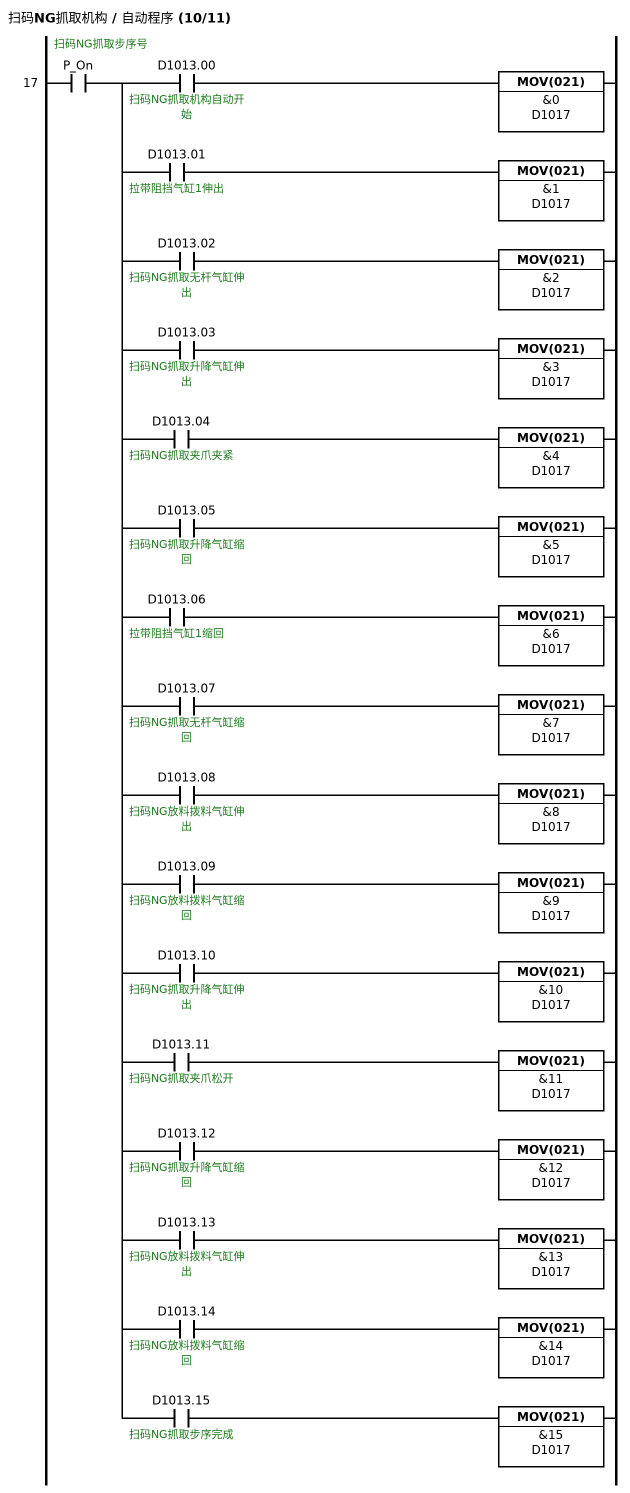
; rung 17: 扫码NG抓取步序号
LD P_On
OUT TR0
AND D1013.00  ; 扫码NG抓取机构自动开始
MOV(021) &0 D1017
LD TR0
AND D1013.01  ; 拉带阻挡气缸1伸出
MOV(021) &1 D1017
LD TR0
AND D1013.02  ; 扫码NG抓取无杆气缸伸出
MOV(021) &2 D1017
LD TR0
AND D1013.03  ; 扫码NG抓取升降气缸伸出
MOV(021) &3 D1017
LD TR0
AND D1013.04  ; 扫码NG抓取夹爪夹紧
MOV(021) &4 D1017
LD TR0
AND D1013.05  ; 扫码NG抓取升降气缸缩回
MOV(021) &5 D1017
LD TR0
AND D1013.06  ; 拉带阻挡气缸1缩回
MOV(021) &6 D1017
LD TR0
AND D1013.07  ; 扫码NG抓取无杆气缸缩回
MOV(021) &7 D1017
LD TR0
AND D1013.08  ; 扫码NG放料拨料气缸伸出
MOV(021) &8 D1017
LD TR0
AND D1013.09  ; 扫码NG放料拨料气缸缩回
MOV(021) &9 D1017
LD TR0
AND D1013.10  ; 扫码NG抓取升降气缸伸出
MOV(021) &10 D1017
LD TR0
AND D1013.11  ; 扫码NG抓取夹爪松开
MOV(021) &11 D1017
LD TR0
AND D1013.12  ; 扫码NG抓取升降气缸缩回
MOV(021) &12 D1017
LD TR0
AND D1013.13  ; 扫码NG放料拨料气缸伸出
MOV(021) &13 D1017
LD TR0
AND D1013.14  ; 扫码NG放料拨料气缸缩回
MOV(021) &14 D1017
LD TR0
AND D1013.15  ; 扫码NG抓取步序完成
MOV(021) &15 D1017

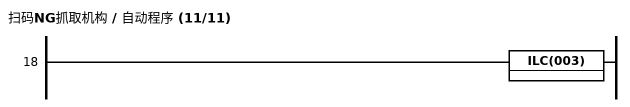
; rung 18
ILC(003)

### Section 状态指示灯

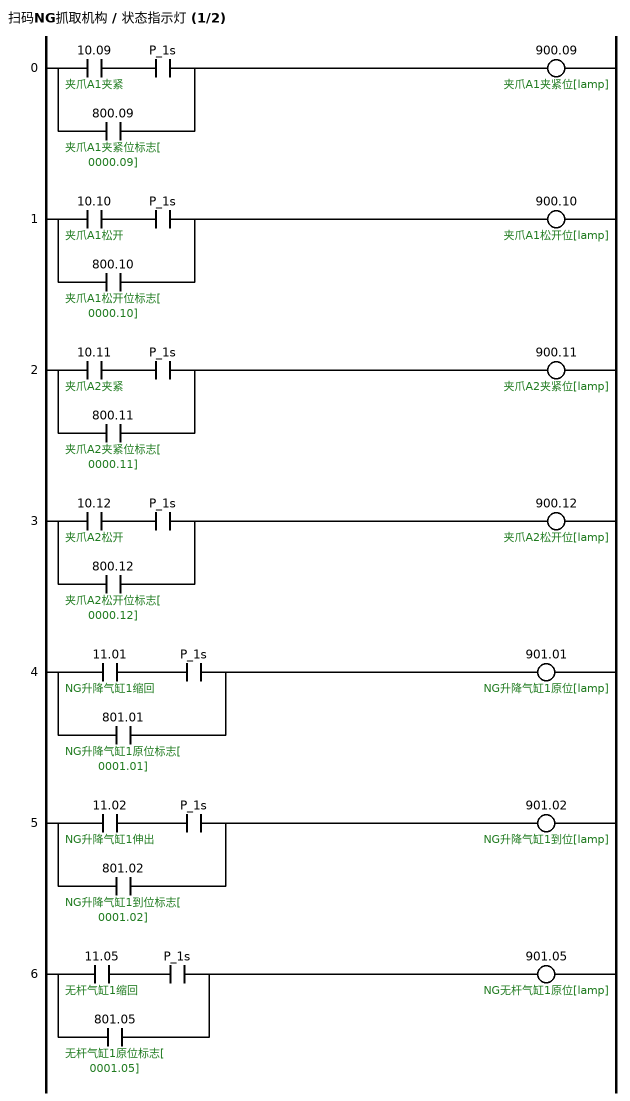
; rung 0
LD 10.09  ; 夹爪A1夹紧
AND P_1s
OR 800.09  ; 夹爪A1夹紧位标志[0000.09]
OUT 900.09  ; 夹爪A1夹紧位[lamp]
; rung 1
LD 10.10  ; 夹爪A1松开
AND P_1s
OR 800.10  ; 夹爪A1松开位标志[0000.10]
OUT 900.10  ; 夹爪A1松开位[lamp]
; rung 2
LD 10.11  ; 夹爪A2夹紧
AND P_1s
OR 800.11  ; 夹爪A2夹紧位标志[0000.11]
OUT 900.11  ; 夹爪A2夹紧位[lamp]
; rung 3
LD 10.12  ; 夹爪A2松开
AND P_1s
OR 800.12  ; 夹爪A2松开位标志[0000.12]
OUT 900.12  ; 夹爪A2松开位[lamp]
; rung 4
LD 11.01  ; NG升降气缸1缩回
AND P_1s
OR 801.01  ; NG升降气缸1原位标志[0001.01]
OUT 901.01  ; NG升降气缸1原位[lamp]
; rung 5
LD 11.02  ; NG升降气缸1伸出
AND P_1s
OR 801.02  ; NG升降气缸1到位标志[0001.02]
OUT 901.02  ; NG升降气缸1到位[lamp]
; rung 6
LD 11.05  ; 无杆气缸1缩回
AND P_1s
OR 801.05  ; 无杆气缸1原位标志[0001.05]
OUT 901.05  ; NG无杆气缸1原位[lamp]

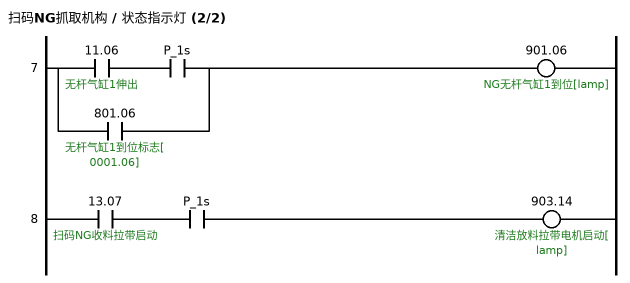
; rung 7
LD 11.06  ; 无杆气缸1伸出
AND P_1s
OR 801.06  ; 无杆气缸1到位标志[0001.06]
OUT 901.06  ; NG无杆气缸1到位[lamp]
; rung 8
LD 13.07  ; 扫码NG收料拉带启动
AND P_1s
OUT 903.14  ; 清洁放料拉带电机启动[lamp]

### Section 输出程序

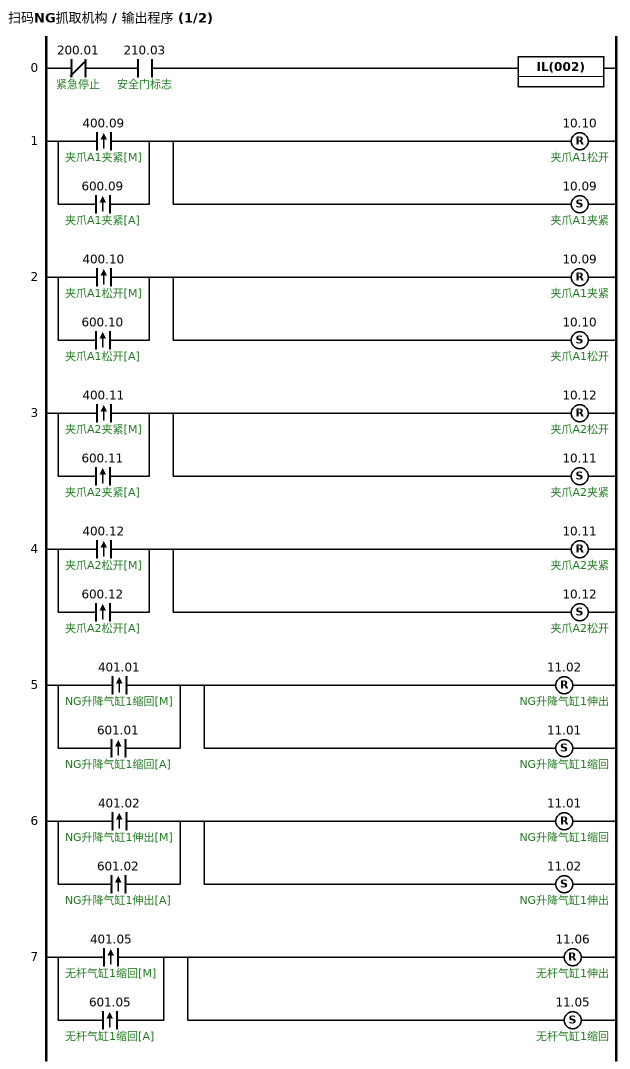
; rung 0
LDNOT 200.01  ; 紧急停止
AND 210.03  ; 安全门标志
IL(002)
; rung 1
@LD 400.09  ; 夹爪A1夹紧[M]
@OR 600.09  ; 夹爪A1夹紧[A]
RSET 10.10  ; 夹爪A1松开
SET 10.09  ; 夹爪A1夹紧
; rung 2
@LD 400.10  ; 夹爪A1松开[M]
@OR 600.10  ; 夹爪A1松开[A]
RSET 10.09  ; 夹爪A1夹紧
SET 10.10  ; 夹爪A1松开
; rung 3
@LD 400.11  ; 夹爪A2夹紧[M]
@OR 600.11  ; 夹爪A2夹紧[A]
RSET 10.12  ; 夹爪A2松开
SET 10.11  ; 夹爪A2夹紧
; rung 4
@LD 400.12  ; 夹爪A2松开[M]
@OR 600.12  ; 夹爪A2松开[A]
RSET 10.11  ; 夹爪A2夹紧
SET 10.12  ; 夹爪A2松开
; rung 5
@LD 401.01  ; NG升降气缸1缩回[M]
@OR 601.01  ; NG升降气缸1缩回[A]
RSET 11.02  ; NG升降气缸1伸出
SET 11.01  ; NG升降气缸1缩回
; rung 6
@LD 401.02  ; NG升降气缸1伸出[M]
@OR 601.02  ; NG升降气缸1伸出[A]
RSET 11.01  ; NG升降气缸1缩回
SET 11.02  ; NG升降气缸1伸出
; rung 7
@LD 401.05  ; 无杆气缸1缩回[M]
@OR 601.05  ; 无杆气缸1缩回[A]
RSET 11.06  ; 无杆气缸1伸出
SET 11.05  ; 无杆气缸1缩回

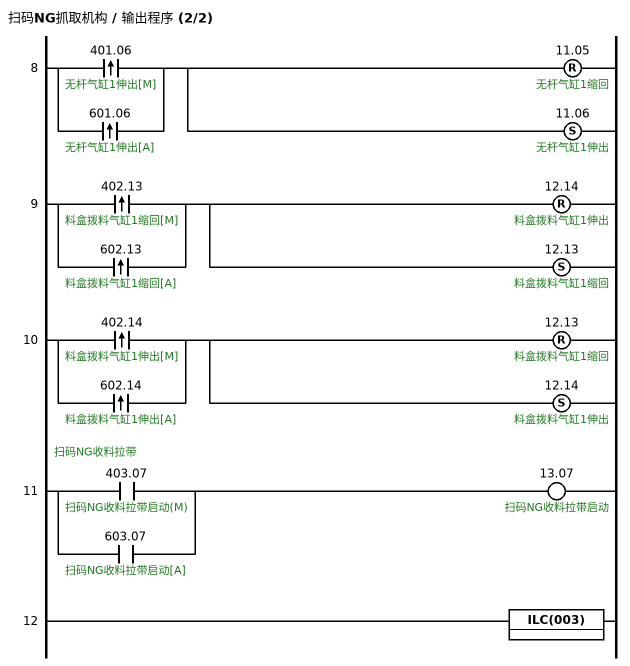
; rung 8
@LD 401.06  ; 无杆气缸1伸出[M]
@OR 601.06  ; 无杆气缸1伸出[A]
RSET 11.05  ; 无杆气缸1缩回
SET 11.06  ; 无杆气缸1伸出
; rung 9
@LD 402.13  ; 料盒拨料气缸1缩回[M]
@OR 602.13  ; 料盒拨料气缸1缩回[A]
RSET 12.14  ; 料盒拨料气缸1伸出
SET 12.13  ; 料盒拨料气缸1缩回
; rung 10
@LD 402.14  ; 料盒拨料气缸1伸出[M]
@OR 602.14  ; 料盒拨料气缸1伸出[A]
RSET 12.13  ; 料盒拨料气缸1缩回
SET 12.14  ; 料盒拨料气缸1伸出
; rung 11: 扫码NG收料拉带
LD 403.07  ; 扫码NG收料拉带启动(M)
OR 603.07  ; 扫码NG收料拉带启动[A]
OUT 13.07  ; 扫码NG收料拉带启动
; rung 12
ILC(003)

### Section END
; rung 0
END(001)

## Program 电池清洁机构 (cyclic task 3)

### Section 主程序

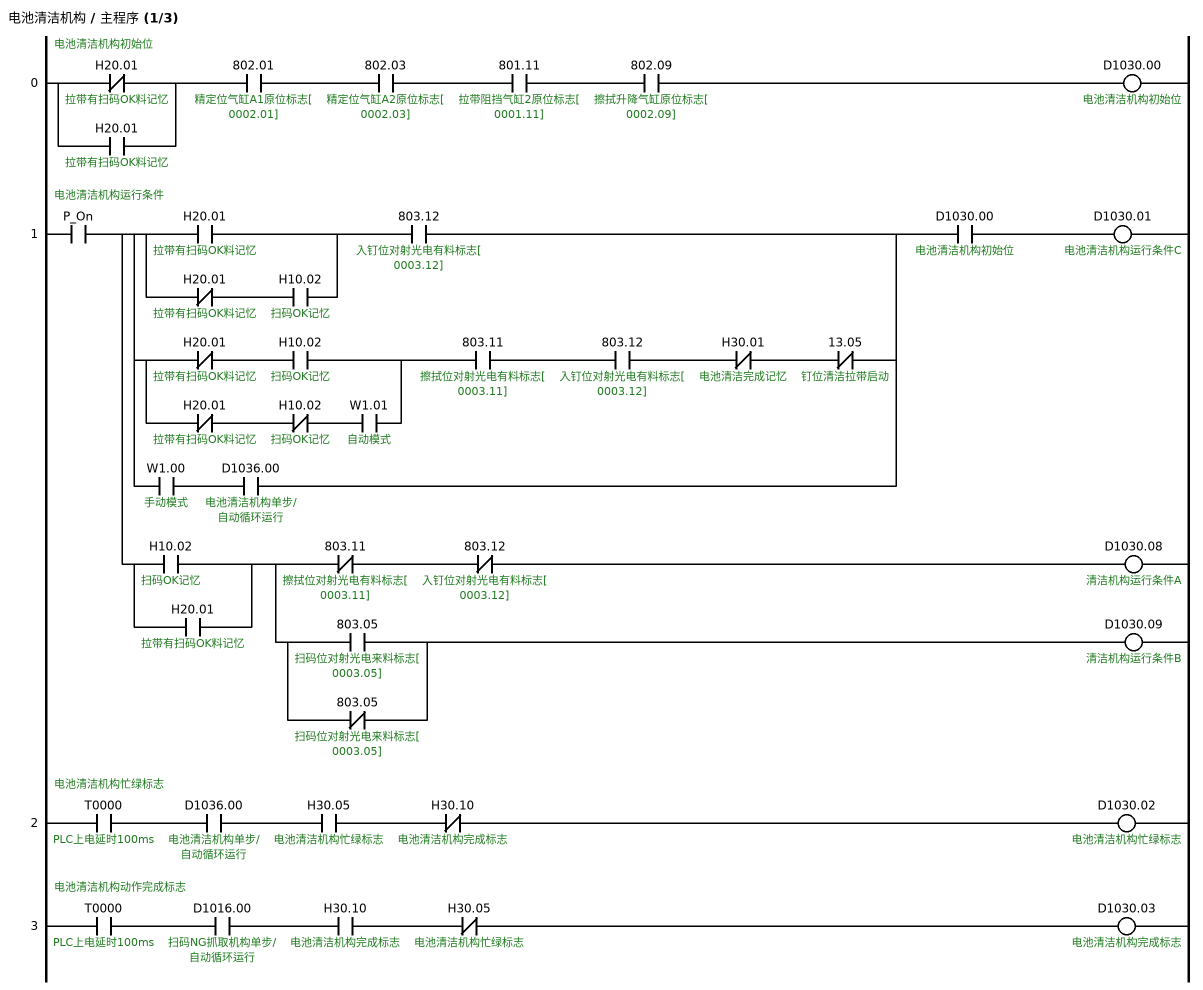
; rung 0: 电池清洁机构初始位
LDNOT H20.01  ; 拉带有扫码OK料记忆
OR H20.01  ; 拉带有扫码OK料记忆
AND 802.01  ; 精定位气缸A1原位标志[0002.01]
AND 802.03  ; 精定位气缸A2原位标志[0002.03]
AND 801.11  ; 拉带阻挡气缸2原位标志[0001.11]
AND 802.09  ; 擦拭升降气缸原位标志[0002.09]
OUT D1030.00  ; 电池清洁机构初始位
; rung 1: 电池清洁机构运行条件
LD P_On
OUT TR0
LD H20.01  ; 拉带有扫码OK料记忆
LDNOT H20.01  ; 拉带有扫码OK料记忆
AND H10.02  ; 扫码OK记忆
ORLD
AND 803.12  ; 入钉位对射光电有料标志[0003.12]
LDNOT H20.01  ; 拉带有扫码OK料记忆
AND H10.02  ; 扫码OK记忆
LDNOT H20.01  ; 拉带有扫码OK料记忆
ANDNOT H10.02  ; 扫码OK记忆
AND W1.01  ; 自动模式
ORLD
AND 803.11  ; 擦拭位对射光电有料标志[0003.11]
AND 803.12  ; 入钉位对射光电有料标志[0003.12]
ANDNOT H30.01  ; 电池清洁完成记忆
ANDNOT 13.05  ; 钉位清洁拉带启动
ORLD
LD W1.00  ; 手动模式
AND D1036.00  ; 电池清洁机构单步/自动循环运行
ORLD
ANDLD
AND D1030.00  ; 电池清洁机构初始位
OUT D1030.01  ; 电池清洁机构运行条件C
LD TR0
LD H10.02  ; 扫码OK记忆
OR H20.01  ; 拉带有扫码OK料记忆
ANDLD
OUT TR0
ANDNOT 803.11  ; 擦拭位对射光电有料标志[0003.11]
ANDNOT 803.12  ; 入钉位对射光电有料标志[0003.12]
OUT D1030.08  ; 清洁机构运行条件A
LD TR0
LD 803.05  ; 扫码位对射光电来料标志[0003.05]
ORNOT 803.05  ; 扫码位对射光电来料标志[0003.05]
ANDLD
OUT D1030.09  ; 清洁机构运行条件B
; rung 2: 电池清洁机构忙绿标志
LD T0000  ; PLC上电延时100ms
AND D1036.00  ; 电池清洁机构单步/自动循环运行
AND H30.05  ; 电池清洁机构忙绿标志
ANDNOT H30.10  ; 电池清洁机构完成标志
OUT D1030.02  ; 电池清洁机构忙绿标志
; rung 3: 电池清洁机构动作完成标志
LD T0000  ; PLC上电延时100ms
AND D1016.00  ; 扫码NG抓取机构单步/自动循环运行
AND H30.10  ; 电池清洁机构完成标志
ANDNOT H30.05  ; 电池清洁机构忙绿标志
OUT D1030.03  ; 电池清洁机构完成标志

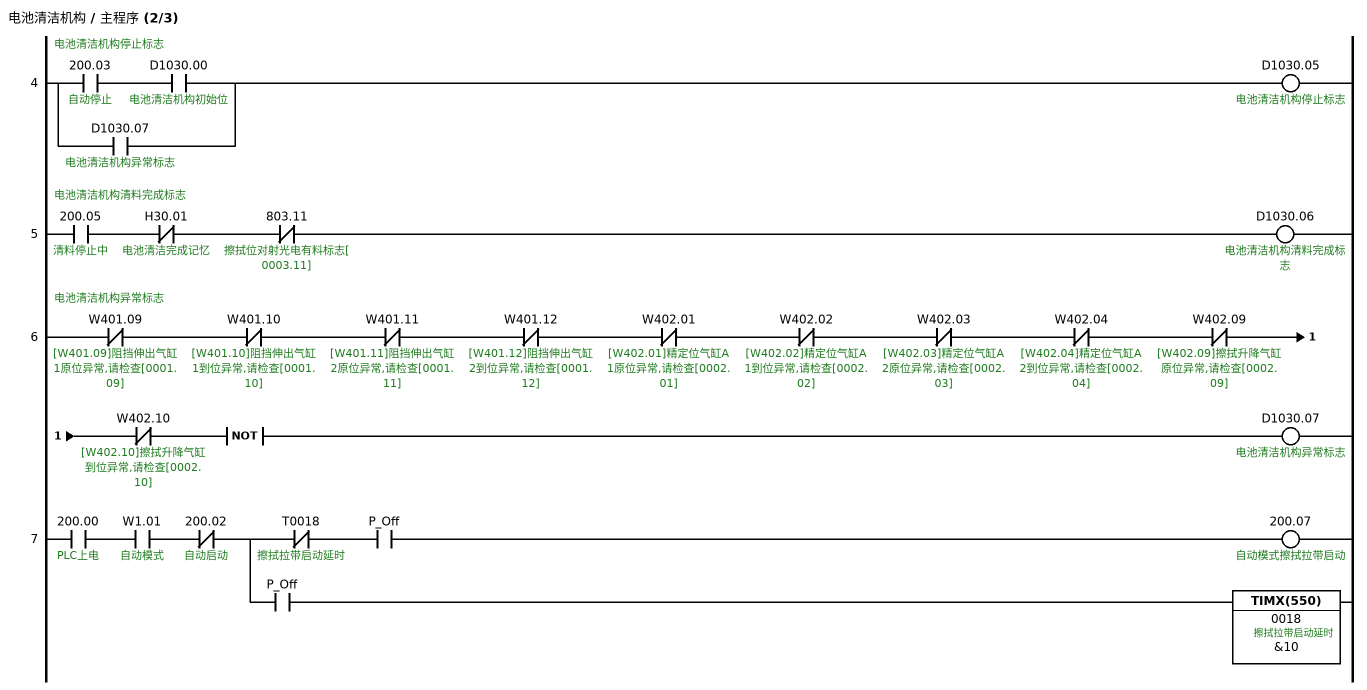
; rung 4: 电池清洁机构停止标志
LD 200.03  ; 自动停止
AND D1030.00  ; 电池清洁机构初始位
OR D1030.07  ; 电池清洁机构异常标志
OUT D1030.05  ; 电池清洁机构停止标志
; rung 5: 电池清洁机构清料完成标志
LD 200.05  ; 清料停止中
ANDNOT H30.01  ; 电池清洁完成记忆
ANDNOT 803.11  ; 擦拭位对射光电有料标志[0003.11]
OUT D1030.06  ; 电池清洁机构清料完成标志
; rung 6: 电池清洁机构异常标志
LDNOT W401.09  ; [W401.09]阻挡伸出气缸1原位异常,请检查[0001.09]
ANDNOT W401.10  ; [W401.10]阻挡伸出气缸1到位异常,请检查[0001.10]
ANDNOT W401.11  ; [W401.11]阻挡伸出气缸2原位异常,请检查[0001.11]
ANDNOT W401.12  ; [W401.12]阻挡伸出气缸2到位异常,请检查[0001.12]
ANDNOT W402.01  ; [W402.01]精定位气缸A1原位异常,请检查[0002.01]
ANDNOT W402.02  ; [W402.02]精定位气缸A1到位异常,请检查[0002.02]
ANDNOT W402.03  ; [W402.03]精定位气缸A2原位异常,请检查[0002.03]
ANDNOT W402.04  ; [W402.04]精定位气缸A2到位异常,请检查[0002.04]
ANDNOT W402.09  ; [W402.09]擦拭升降气缸原位异常,请检查[0002.09]
ANDNOT W402.10  ; [W402.10]擦拭升降气缸到位异常,请检查[0002.10]
NOT(520)
OUT D1030.07  ; 电池清洁机构异常标志
; rung 7
LD 200.00  ; PLC上电
AND W1.01  ; 自动模式
ANDNOT 200.02  ; 自动启动
OUT TR0
ANDNOT T0018  ; 擦拭拉带启动延时
AND P_Off
OUT 200.07  ; 自动模式擦拭拉带启动
LD TR0
AND P_Off
TIMX(550) 0018 &10  ; 擦拭拉带启动延时

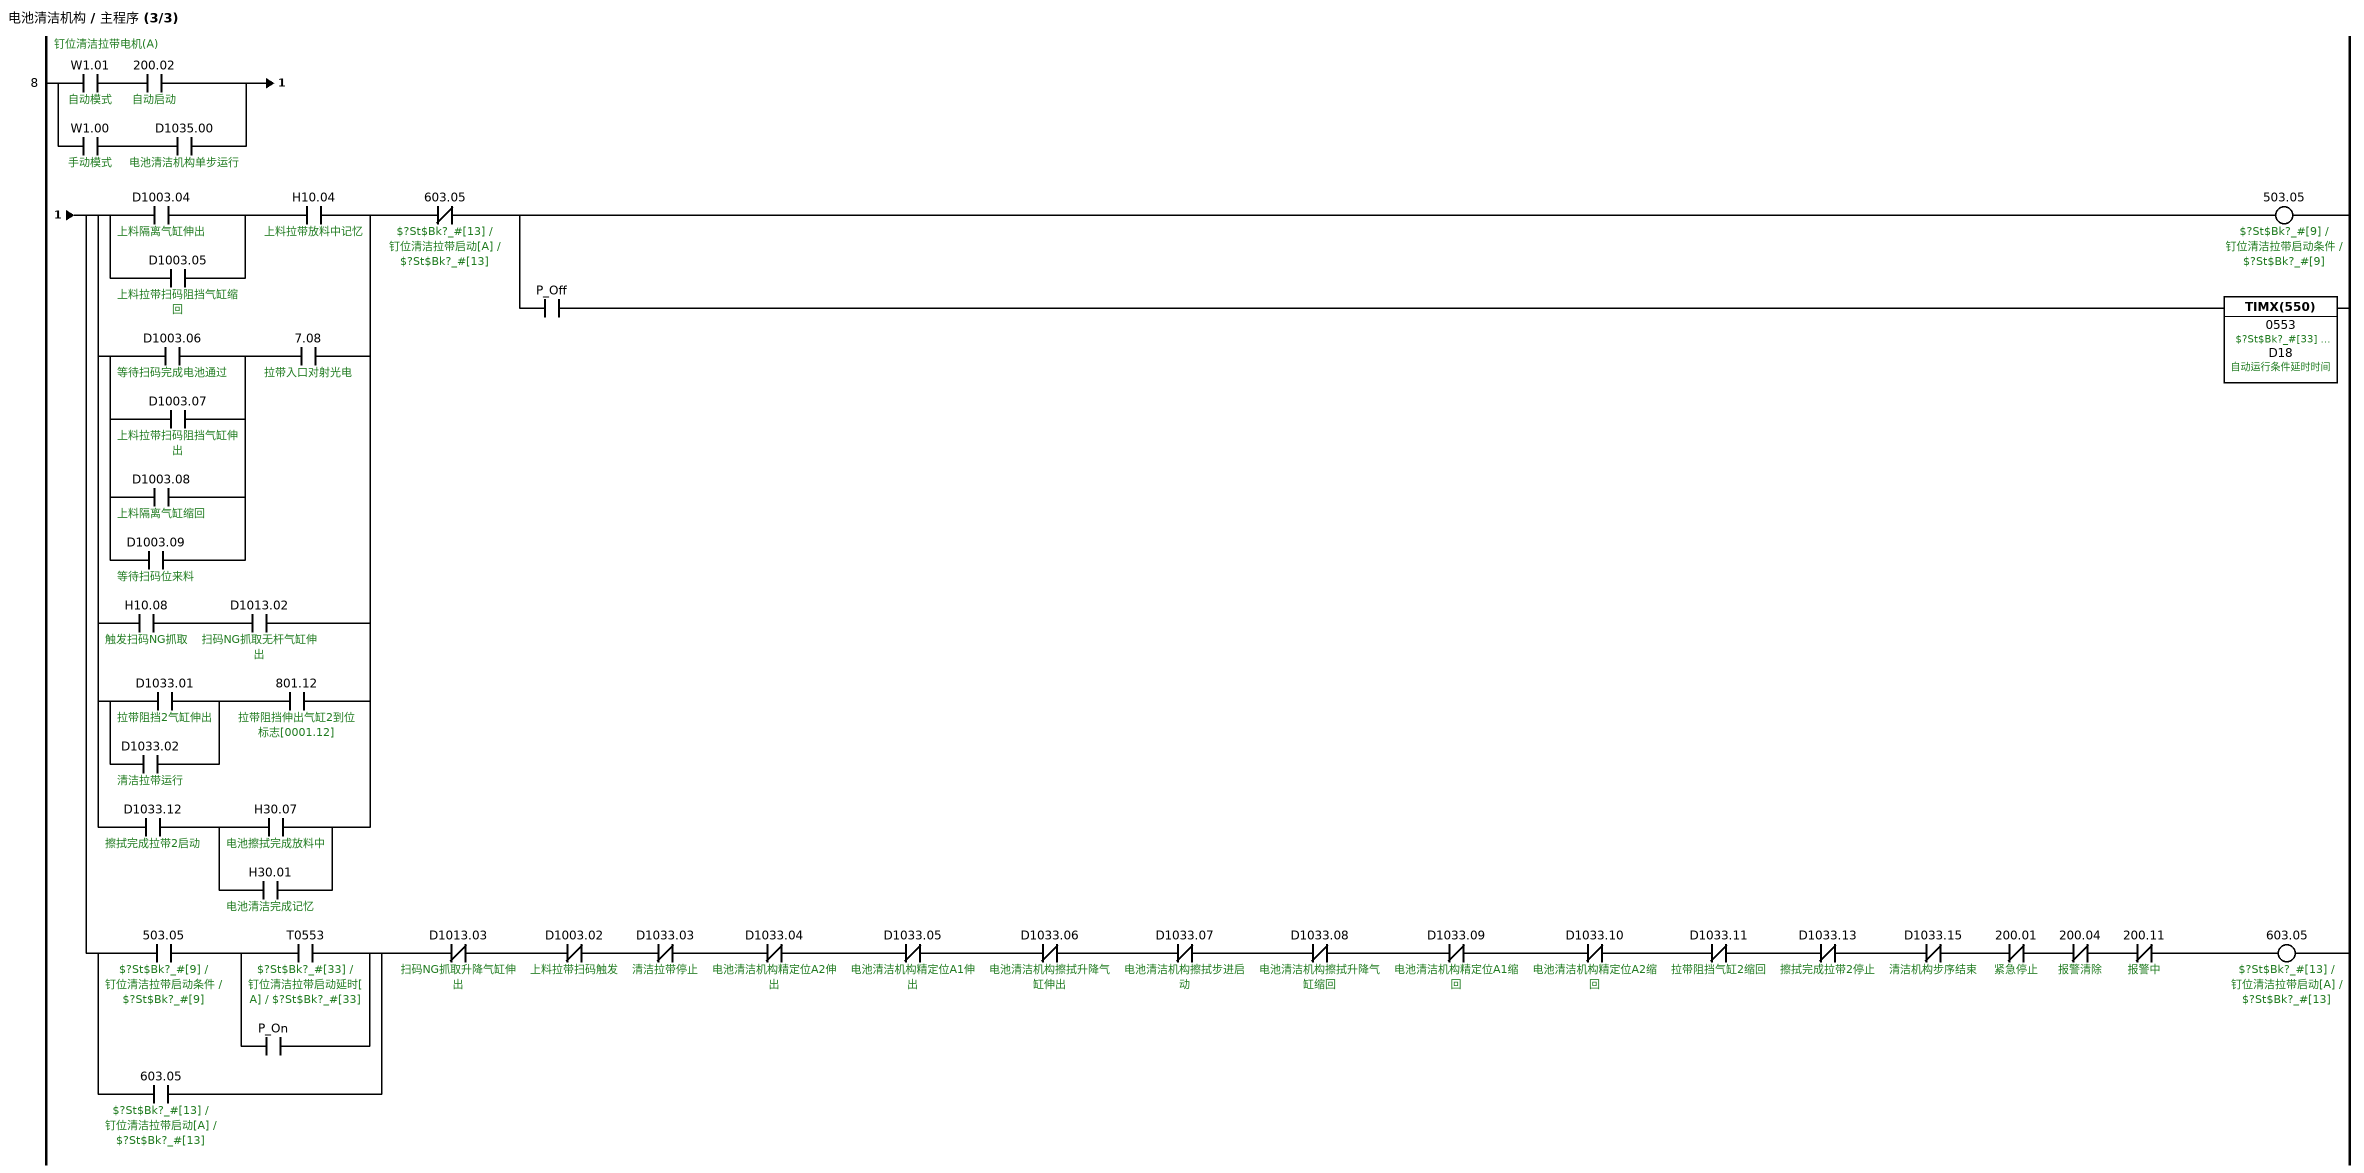
; rung 8: 钉位清洁拉带电机(A)
LD W1.01  ; 自动模式
AND 200.02  ; 自动启动
LD W1.00  ; 手动模式
AND D1035.00  ; 电池清洁机构单步运行
ORLD
OUT TR0
LD D1003.04  ; 上料隔离气缸伸出
OR D1003.05  ; 上料拉带扫码阻挡气缸缩回
AND H10.04  ; 上料拉带放料中记忆
LD D1003.06  ; 等待扫码完成电池通过
OR D1003.07  ; 上料拉带扫码阻挡气缸伸出
OR D1003.08  ; 上料隔离气缸缩回
OR D1003.09  ; 等待扫码位来料
AND 7.08  ; 拉带入口对射光电
ORLD
LD H10.08  ; 触发扫码NG抓取
AND D1013.02  ; 扫码NG抓取无杆气缸伸出
ORLD
LD D1033.01  ; 拉带阻挡2气缸伸出
OR D1033.02  ; 清洁拉带运行
AND 801.12  ; 拉带阻挡伸出气缸2到位标志[0001.12]
ORLD
LD D1033.12  ; 擦拭完成拉带2启动
LD H30.07  ; 电池擦拭完成放料中
OR H30.01  ; 电池清洁完成记忆
ANDLD
ORLD
ANDLD
ANDNOT 603.05  ; $?St$Bk?_#[13] / 钉位清洁拉带启动[A] / $?St$Bk?_#[13]
OUT 503.05  ; $?St$Bk?_#[9] / 钉位清洁拉带启动条件 / $?St$Bk?_#[9]
AND P_Off
TIMX(550) 0553 D18  ; 自动运行条件延时时间, $?St$Bk?_#[33] / 钉位清洁拉带启动延时[A] / $?St$Bk?_#[33]
LD TR0
LD 503.05  ; $?St$Bk?_#[9] / 钉位清洁拉带启动条件 / $?St$Bk?_#[9]
LD T0553  ; $?St$Bk?_#[33] / 钉位清洁拉带启动延时[A] / $?St$Bk?_#[33]
OR P_On
ANDLD
OR 603.05  ; $?St$Bk?_#[13] / 钉位清洁拉带启动[A] / $?St$Bk?_#[13]
ANDLD
ANDNOT D1013.03  ; 扫码NG抓取升降气缸伸出
ANDNOT D1003.02  ; 上料拉带扫码触发
ANDNOT D1033.03  ; 清洁拉带停止
ANDNOT D1033.04  ; 电池清洁机构精定位A2伸出
ANDNOT D1033.05  ; 电池清洁机构精定位A1伸出
ANDNOT D1033.06  ; 电池清洁机构擦拭升降气缸伸出
ANDNOT D1033.07  ; 电池清洁机构擦拭步进启动
ANDNOT D1033.08  ; 电池清洁机构擦拭升降气缸缩回
ANDNOT D1033.09  ; 电池清洁机构精定位A1缩回
ANDNOT D1033.10  ; 电池清洁机构精定位A2缩回
ANDNOT D1033.11  ; 拉带阻挡气缸2缩回
ANDNOT D1033.13  ; 擦拭完成拉带2停止
ANDNOT D1033.15  ; 清洁机构步序结束
ANDNOT 200.01  ; 紧急停止
ANDNOT 200.04  ; 报警清除
ANDNOT 200.11  ; 报警中
OUT 603.05  ; $?St$Bk?_#[13] / 钉位清洁拉带启动[A] / $?St$Bk?_#[13]

### Section 工站复位

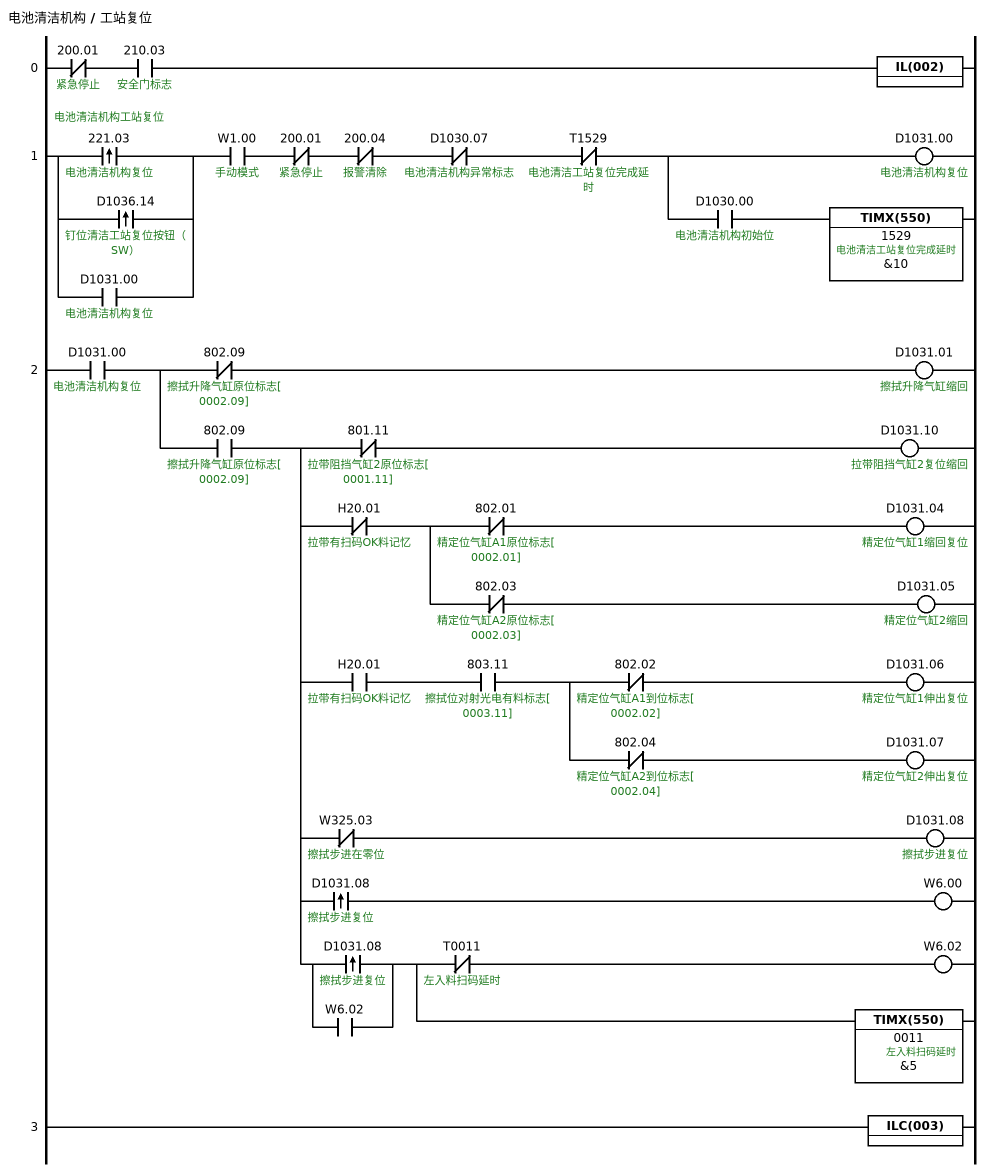
; rung 0
LDNOT 200.01  ; 紧急停止
AND 210.03  ; 安全门标志
IL(002)
; rung 1: 电池清洁机构工站复位
@LD 221.03  ; 电池清洁机构复位
@OR D1036.14  ; 钉位清洁工站复位按钮（SW）
OR D1031.00  ; 电池清洁机构复位
AND W1.00  ; 手动模式
ANDNOT 200.01  ; 紧急停止
ANDNOT 200.04  ; 报警清除
ANDNOT D1030.07  ; 电池清洁机构异常标志
ANDNOT T1529  ; 电池清洁工站复位完成延时
OUT D1031.00  ; 电池清洁机构复位
AND D1030.00  ; 电池清洁机构初始位
TIMX(550) 1529 &10  ; 电池清洁工站复位完成延时
; rung 2
LD D1031.00  ; 电池清洁机构复位
OUT TR0
ANDNOT 802.09  ; 擦拭升降气缸原位标志[0002.09]
OUT D1031.01  ; 擦拭升降气缸缩回
LD TR0
AND 802.09  ; 擦拭升降气缸原位标志[0002.09]
OUT TR0
ANDNOT 801.11  ; 拉带阻挡气缸2原位标志[0001.11]
OUT D1031.10  ; 拉带阻挡气缸2复位缩回
LD TR0
ANDNOT H20.01  ; 拉带有扫码OK料记忆
OUT TR1
ANDNOT 802.01  ; 精定位气缸A1原位标志[0002.01]
OUT D1031.04  ; 精定位气缸1缩回复位
LD TR1
ANDNOT 802.03  ; 精定位气缸A2原位标志[0002.03]
OUT D1031.05  ; 精定位气缸2缩回
LD TR0
AND H20.01  ; 拉带有扫码OK料记忆
AND 803.11  ; 擦拭位对射光电有料标志[0003.11]
OUT TR1
ANDNOT 802.02  ; 精定位气缸A1到位标志[0002.02]
OUT D1031.06  ; 精定位气缸1伸出复位
LD TR1
ANDNOT 802.04  ; 精定位气缸A2到位标志[0002.04]
OUT D1031.07  ; 精定位气缸2伸出复位
LD TR0
ANDNOT W325.03  ; 擦拭步进在零位
OUT D1031.08  ; 擦拭步进复位
LD TR0
@AND D1031.08  ; 擦拭步进复位
OUT W6.00
LD TR0
@LD D1031.08  ; 擦拭步进复位
OR W6.02
ANDLD
OUT TR0
ANDNOT T0011  ; 左入料扫码延时
OUT W6.02
LD TR0
TIMX(550) 0011 &5  ; 左入料扫码延时
; rung 3
ILC(003)

### Section 手动程序

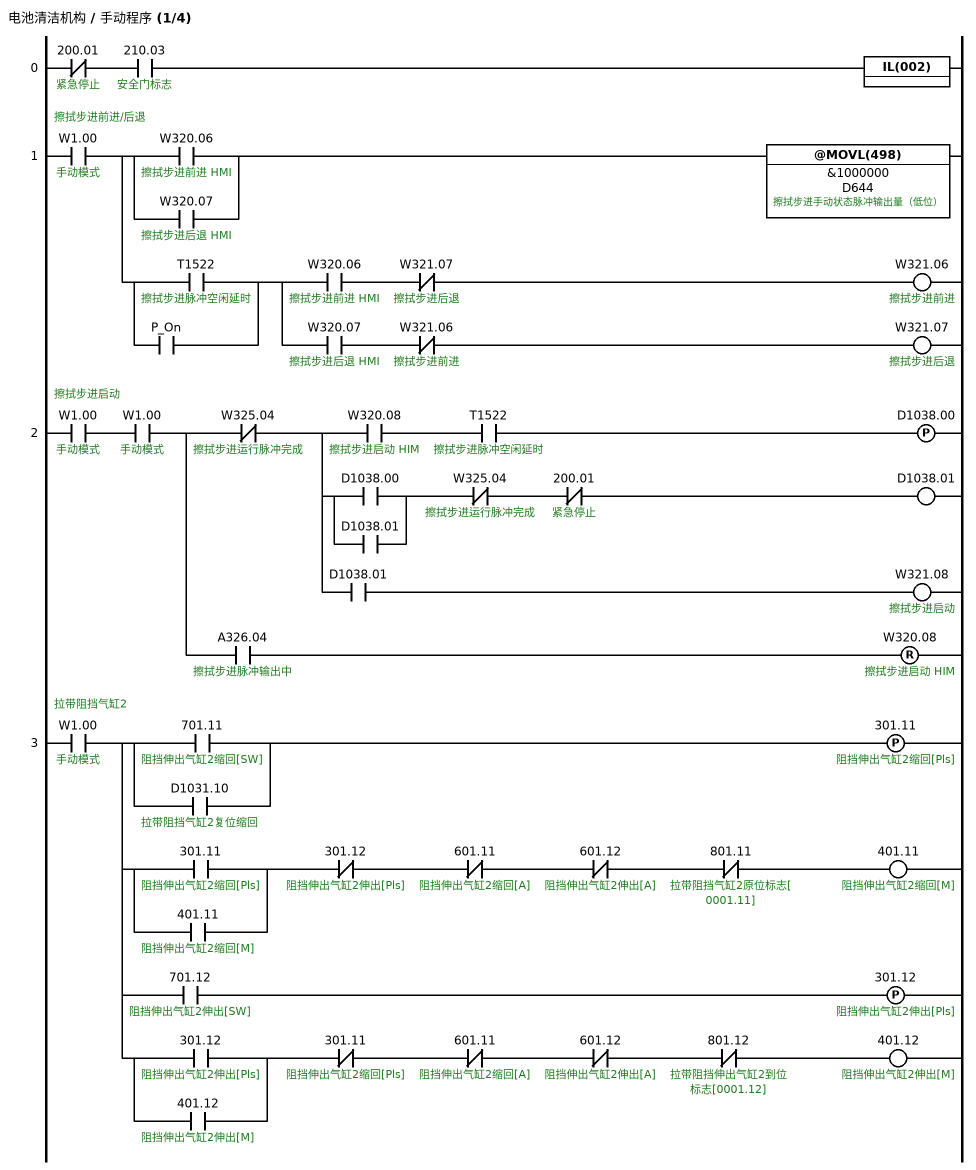
; rung 0
LDNOT 200.01  ; 紧急停止
AND 210.03  ; 安全门标志
IL(002)
; rung 1: 擦拭步进前进/后退
LD W1.00  ; 手动模式
OUT TR0
LD W320.06  ; 擦拭步进前进 HMI
OR W320.07  ; 擦拭步进后退 HMI
ANDLD
@MOVL(498) &1000000 D644  ; 擦拭步进手动状态脉冲输出量（低位）
LD TR0
LD T1522  ; 擦拭步进脉冲空闲延时
OR P_On
ANDLD
OUT TR0
AND W320.06  ; 擦拭步进前进 HMI
ANDNOT W321.07  ; 擦拭步进后退
OUT W321.06  ; 擦拭步进前进
LD TR0
AND W320.07  ; 擦拭步进后退 HMI
ANDNOT W321.06  ; 擦拭步进前进
OUT W321.07  ; 擦拭步进后退
; rung 2: 擦拭步进启动
LD W1.00  ; 手动模式
AND W1.00  ; 手动模式
OUT TR0
ANDNOT W325.04  ; 擦拭步进运行脉冲完成
OUT TR1
AND W320.08  ; 擦拭步进启动 HIM
AND T1522  ; 擦拭步进脉冲空闲延时
DIFU(013) D1038.00
LD TR1
LD D1038.00
OR D1038.01
ANDLD
ANDNOT W325.04  ; 擦拭步进运行脉冲完成
ANDNOT 200.01  ; 紧急停止
OUT D1038.01
LD TR1
AND D1038.01
OUT W321.08  ; 擦拭步进启动
LD TR0
AND A326.04  ; 擦拭步进脉冲输出中
RSET W320.08  ; 擦拭步进启动 HIM
; rung 3: 拉带阻挡气缸2
LD W1.00  ; 手动模式
OUT TR0
LD 701.11  ; 阻挡伸出气缸2缩回[SW]
OR D1031.10  ; 拉带阻挡气缸2复位缩回
ANDLD
DIFU(013) 301.11  ; 阻挡伸出气缸2缩回[Pls]
LD TR0
LD 301.11  ; 阻挡伸出气缸2缩回[Pls]
OR 401.11  ; 阻挡伸出气缸2缩回[M]
ANDLD
ANDNOT 301.12  ; 阻挡伸出气缸2伸出[Pls]
ANDNOT 601.11  ; 阻挡伸出气缸2缩回[A]
ANDNOT 601.12  ; 阻挡伸出气缸2伸出[A]
ANDNOT 801.11  ; 拉带阻挡气缸2原位标志[0001.11]
OUT 401.11  ; 阻挡伸出气缸2缩回[M]
LD TR0
AND 701.12  ; 阻挡伸出气缸2伸出[SW]
DIFU(013) 301.12  ; 阻挡伸出气缸2伸出[Pls]
LD TR0
LD 301.12  ; 阻挡伸出气缸2伸出[Pls]
OR 401.12  ; 阻挡伸出气缸2伸出[M]
ANDLD
ANDNOT 301.11  ; 阻挡伸出气缸2缩回[Pls]
ANDNOT 601.11  ; 阻挡伸出气缸2缩回[A]
ANDNOT 601.12  ; 阻挡伸出气缸2伸出[A]
ANDNOT 801.12  ; 拉带阻挡伸出气缸2到位标志[0001.12]
OUT 401.12  ; 阻挡伸出气缸2伸出[M]

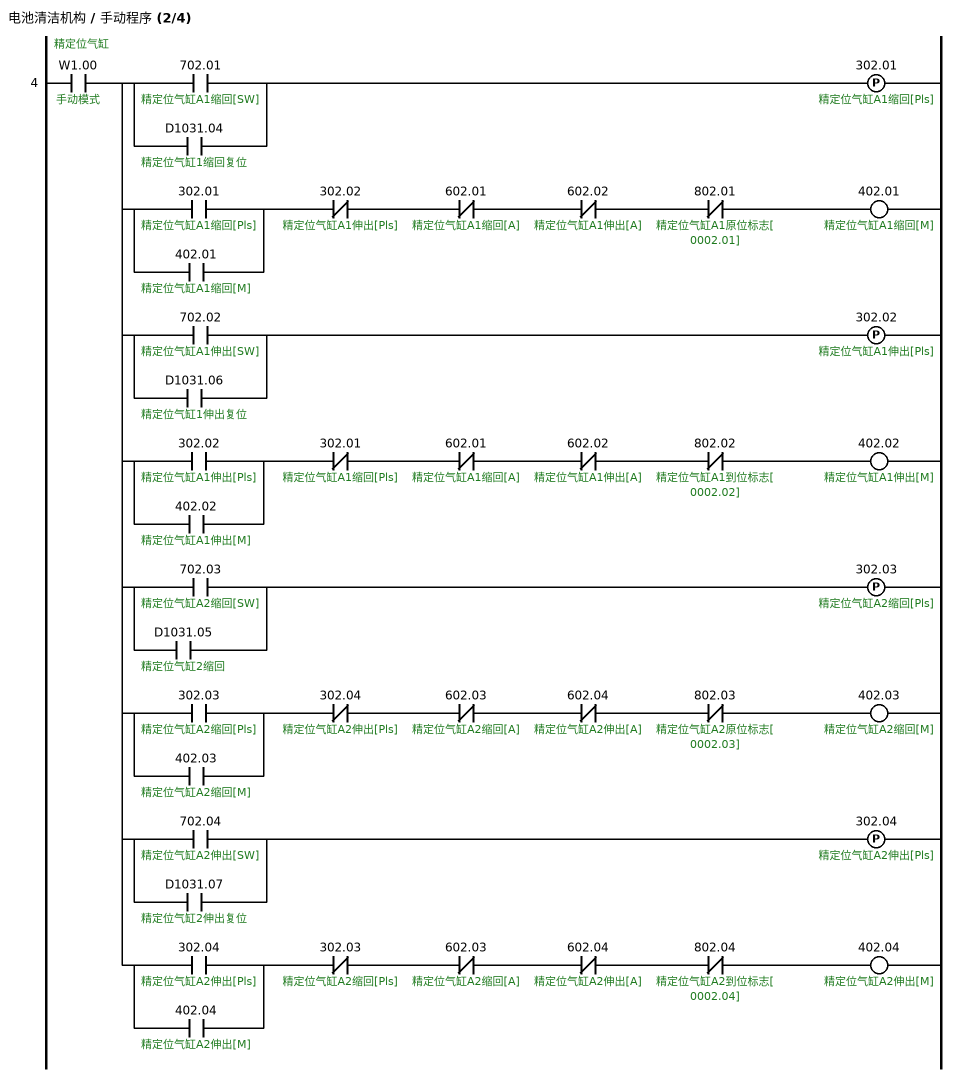
; rung 4: 精定位气缸
LD W1.00  ; 手动模式
OUT TR0
LD 702.01  ; 精定位气缸A1缩回[SW]
OR D1031.04  ; 精定位气缸1缩回复位
ANDLD
DIFU(013) 302.01  ; 精定位气缸A1缩回[Pls]
LD TR0
LD 302.01  ; 精定位气缸A1缩回[Pls]
OR 402.01  ; 精定位气缸A1缩回[M]
ANDLD
ANDNOT 302.02  ; 精定位气缸A1伸出[Pls]
ANDNOT 602.01  ; 精定位气缸A1缩回[A]
ANDNOT 602.02  ; 精定位气缸A1伸出[A]
ANDNOT 802.01  ; 精定位气缸A1原位标志[0002.01]
OUT 402.01  ; 精定位气缸A1缩回[M]
LD TR0
LD 702.02  ; 精定位气缸A1伸出[SW]
OR D1031.06  ; 精定位气缸1伸出复位
ANDLD
DIFU(013) 302.02  ; 精定位气缸A1伸出[Pls]
LD TR0
LD 302.02  ; 精定位气缸A1伸出[Pls]
OR 402.02  ; 精定位气缸A1伸出[M]
ANDLD
ANDNOT 302.01  ; 精定位气缸A1缩回[Pls]
ANDNOT 602.01  ; 精定位气缸A1缩回[A]
ANDNOT 602.02  ; 精定位气缸A1伸出[A]
ANDNOT 802.02  ; 精定位气缸A1到位标志[0002.02]
OUT 402.02  ; 精定位气缸A1伸出[M]
LD TR0
LD 702.03  ; 精定位气缸A2缩回[SW]
OR D1031.05  ; 精定位气缸2缩回
ANDLD
DIFU(013) 302.03  ; 精定位气缸A2缩回[Pls]
LD TR0
LD 302.03  ; 精定位气缸A2缩回[Pls]
OR 402.03  ; 精定位气缸A2缩回[M]
ANDLD
ANDNOT 302.04  ; 精定位气缸A2伸出[Pls]
ANDNOT 602.03  ; 精定位气缸A2缩回[A]
ANDNOT 602.04  ; 精定位气缸A2伸出[A]
ANDNOT 802.03  ; 精定位气缸A2原位标志[0002.03]
OUT 402.03  ; 精定位气缸A2缩回[M]
LD TR0
LD 702.04  ; 精定位气缸A2伸出[SW]
OR D1031.07  ; 精定位气缸2伸出复位
ANDLD
DIFU(013) 302.04  ; 精定位气缸A2伸出[Pls]
LD TR0
LD 302.04  ; 精定位气缸A2伸出[Pls]
OR 402.04  ; 精定位气缸A2伸出[M]
ANDLD
ANDNOT 302.03  ; 精定位气缸A2缩回[Pls]
ANDNOT 602.03  ; 精定位气缸A2缩回[A]
ANDNOT 602.04  ; 精定位气缸A2伸出[A]
ANDNOT 802.04  ; 精定位气缸A2到位标志[0002.04]
OUT 402.04  ; 精定位气缸A2伸出[M]

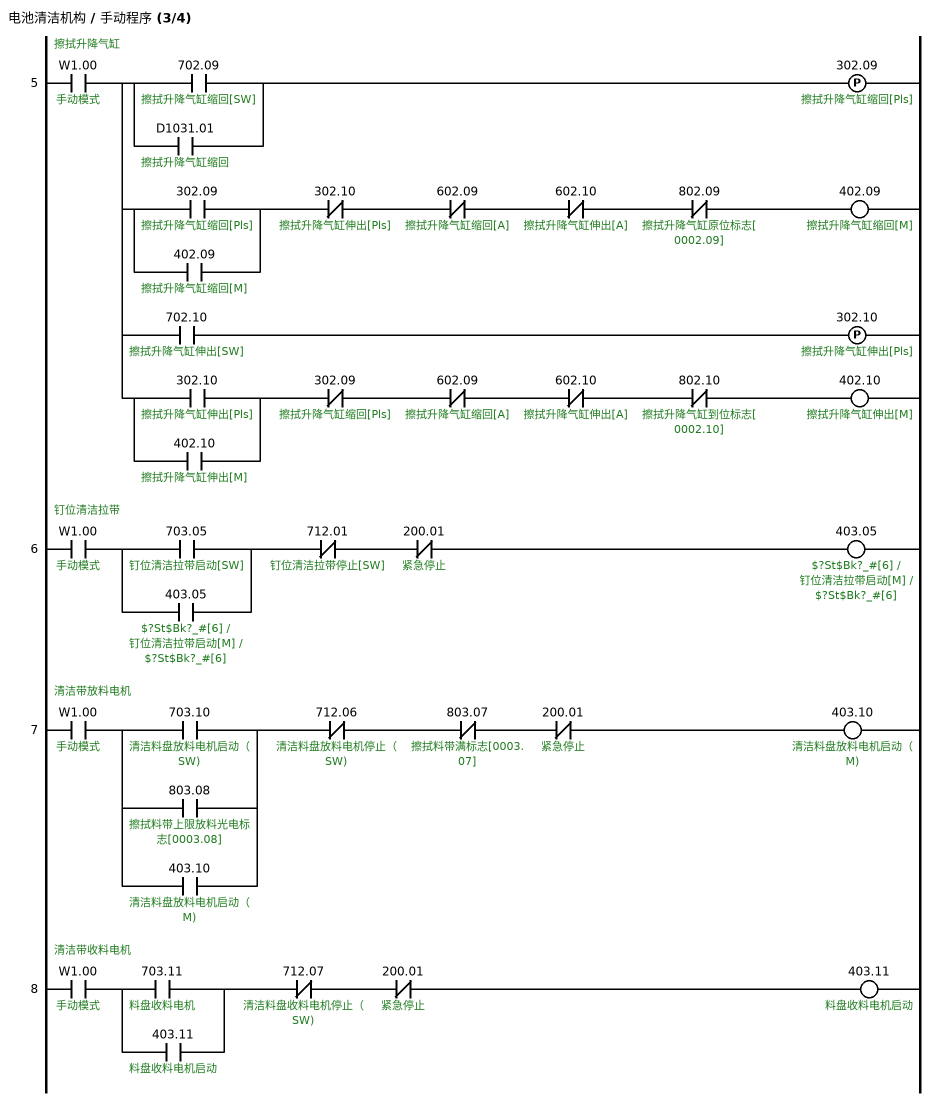
; rung 5: 擦拭升降气缸
LD W1.00  ; 手动模式
OUT TR0
LD 702.09  ; 擦拭升降气缸缩回[SW]
OR D1031.01  ; 擦拭升降气缸缩回
ANDLD
DIFU(013) 302.09  ; 擦拭升降气缸缩回[Pls]
LD TR0
LD 302.09  ; 擦拭升降气缸缩回[Pls]
OR 402.09  ; 擦拭升降气缸缩回[M]
ANDLD
ANDNOT 302.10  ; 擦拭升降气缸伸出[Pls]
ANDNOT 602.09  ; 擦拭升降气缸缩回[A]
ANDNOT 602.10  ; 擦拭升降气缸伸出[A]
ANDNOT 802.09  ; 擦拭升降气缸原位标志[0002.09]
OUT 402.09  ; 擦拭升降气缸缩回[M]
LD TR0
AND 702.10  ; 擦拭升降气缸伸出[SW]
DIFU(013) 302.10  ; 擦拭升降气缸伸出[Pls]
LD TR0
LD 302.10  ; 擦拭升降气缸伸出[Pls]
OR 402.10  ; 擦拭升降气缸伸出[M]
ANDLD
ANDNOT 302.09  ; 擦拭升降气缸缩回[Pls]
ANDNOT 602.09  ; 擦拭升降气缸缩回[A]
ANDNOT 602.10  ; 擦拭升降气缸伸出[A]
ANDNOT 802.10  ; 擦拭升降气缸到位标志[0002.10]
OUT 402.10  ; 擦拭升降气缸伸出[M]
; rung 6: 钉位清洁拉带
LD W1.00  ; 手动模式
LD 703.05  ; 钉位清洁拉带启动[SW]
OR 403.05  ; $?St$Bk?_#[6] / 钉位清洁拉带启动[M] / $?St$Bk?_#[6]
ANDLD
ANDNOT 712.01  ; 钉位清洁拉带停止[SW]
ANDNOT 200.01  ; 紧急停止
OUT 403.05  ; $?St$Bk?_#[6] / 钉位清洁拉带启动[M] / $?St$Bk?_#[6]
; rung 7: 清洁带放料电机
LD W1.00  ; 手动模式
LD 703.10  ; 清洁料盘放料电机启动（SW)
OR 803.08  ; 擦拭料带上限放料光电标志[0003.08]
OR 403.10  ; 清洁料盘放料电机启动（M)
ANDLD
ANDNOT 712.06  ; 清洁料盘放料电机停止（SW)
ANDNOT 803.07  ; 擦拭料带满标志[0003.07]
ANDNOT 200.01  ; 紧急停止
OUT 403.10  ; 清洁料盘放料电机启动（M)
; rung 8: 清洁带收料电机
LD W1.00  ; 手动模式
LD 703.11  ; 料盘收料电机
OR 403.11  ; 料盘收料电机启动
ANDLD
ANDNOT 712.07  ; 清洁料盘收料电机停止（SW)
ANDNOT 200.01  ; 紧急停止
OUT 403.11  ; 料盘收料电机启动

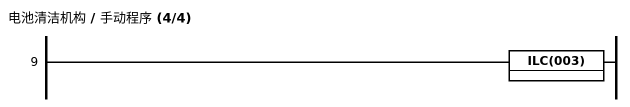
; rung 9
ILC(003)

### Section 自动程序

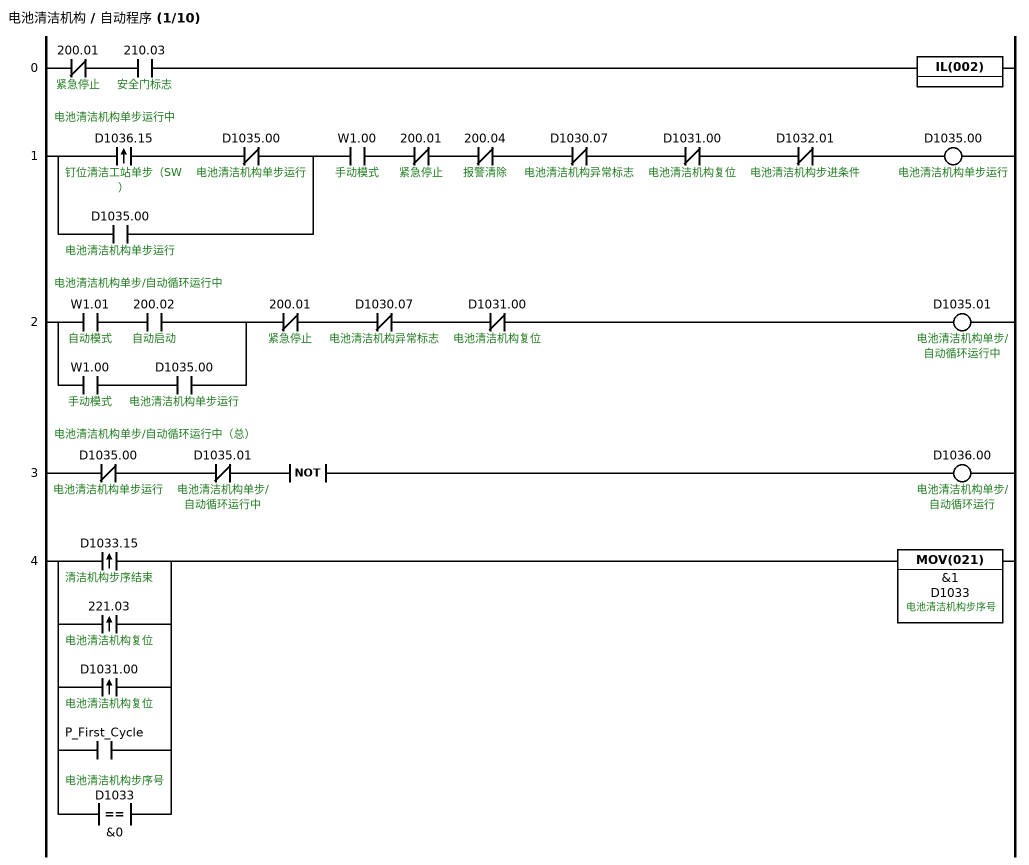
; rung 0
LDNOT 200.01  ; 紧急停止
AND 210.03  ; 安全门标志
IL(002)
; rung 1: 电池清洁机构单步运行中
@LD D1036.15  ; 钉位清洁工站单步（SW）
ANDNOT D1035.00  ; 电池清洁机构单步运行
OR D1035.00  ; 电池清洁机构单步运行
AND W1.00  ; 手动模式
ANDNOT 200.01  ; 紧急停止
ANDNOT 200.04  ; 报警清除
ANDNOT D1030.07  ; 电池清洁机构异常标志
ANDNOT D1031.00  ; 电池清洁机构复位
ANDNOT D1032.01  ; 电池清洁机构步进条件
OUT D1035.00  ; 电池清洁机构单步运行
; rung 2: 电池清洁机构单步/自动循环运行中
LD W1.01  ; 自动模式
AND 200.02  ; 自动启动
LD W1.00  ; 手动模式
AND D1035.00  ; 电池清洁机构单步运行
ORLD
ANDNOT 200.01  ; 紧急停止
ANDNOT D1030.07  ; 电池清洁机构异常标志
ANDNOT D1031.00  ; 电池清洁机构复位
OUT D1035.01  ; 电池清洁机构单步/自动循环运行中
; rung 3: 电池清洁机构单步/自动循环运行中（总）
LDNOT D1035.00  ; 电池清洁机构单步运行
ANDNOT D1035.01  ; 电池清洁机构单步/自动循环运行中
NOT(520)
OUT D1036.00  ; 电池清洁机构单步/自动循环运行
; rung 4
@LD D1033.15  ; 清洁机构步序结束
@OR 221.03  ; 电池清洁机构复位
@OR D1031.00  ; 电池清洁机构复位
OR P_First_Cycle
OR=(300) D1033 &0  ; 电池清洁机构步序号
MOV(021) &1 D1033  ; 电池清洁机构步序号

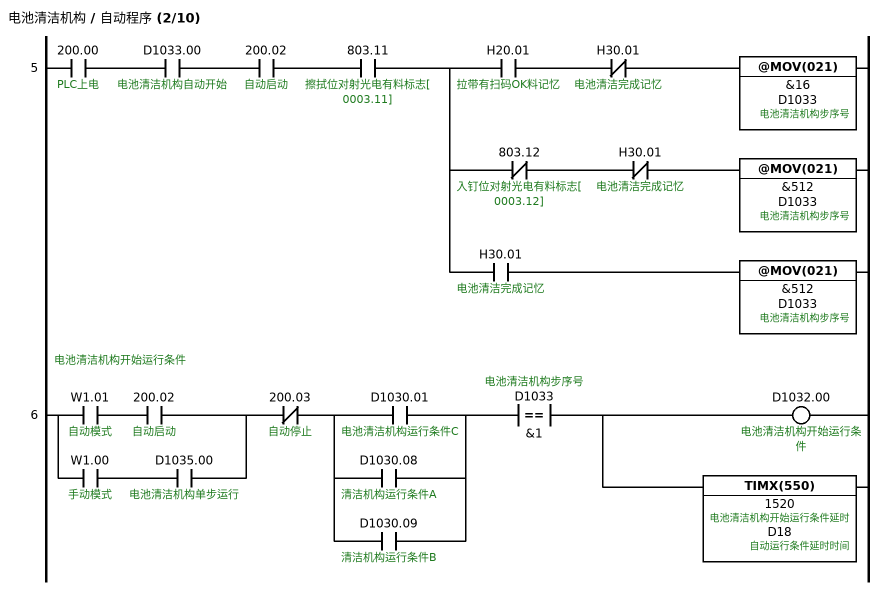
; rung 5
LD 200.00  ; PLC上电
AND D1033.00  ; 电池清洁机构自动开始
AND 200.02  ; 自动启动
AND 803.11  ; 擦拭位对射光电有料标志[0003.11]
OUT TR0
AND H20.01  ; 拉带有扫码OK料记忆
ANDNOT H30.01  ; 电池清洁完成记忆
@MOV(021) &16 D1033  ; 电池清洁机构步序号
LD TR0
ANDNOT 803.12  ; 入钉位对射光电有料标志[0003.12]
ANDNOT H30.01  ; 电池清洁完成记忆
@MOV(021) &512 D1033  ; 电池清洁机构步序号
LD TR0
AND H30.01  ; 电池清洁完成记忆
@MOV(021) &512 D1033  ; 电池清洁机构步序号
; rung 6: 电池清洁机构开始运行条件
LD W1.01  ; 自动模式
AND 200.02  ; 自动启动
LD W1.00  ; 手动模式
AND D1035.00  ; 电池清洁机构单步运行
ORLD
ANDNOT 200.03  ; 自动停止
LD D1030.01  ; 电池清洁机构运行条件C
OR D1030.08  ; 清洁机构运行条件A
OR D1030.09  ; 清洁机构运行条件B
ANDLD
AND=(300) D1033 &1  ; 电池清洁机构步序号
OUT D1032.00  ; 电池清洁机构开始运行条件
TIMX(550) 1520 D18  ; 自动运行条件延时时间, 电池清洁机构开始运行条件延时

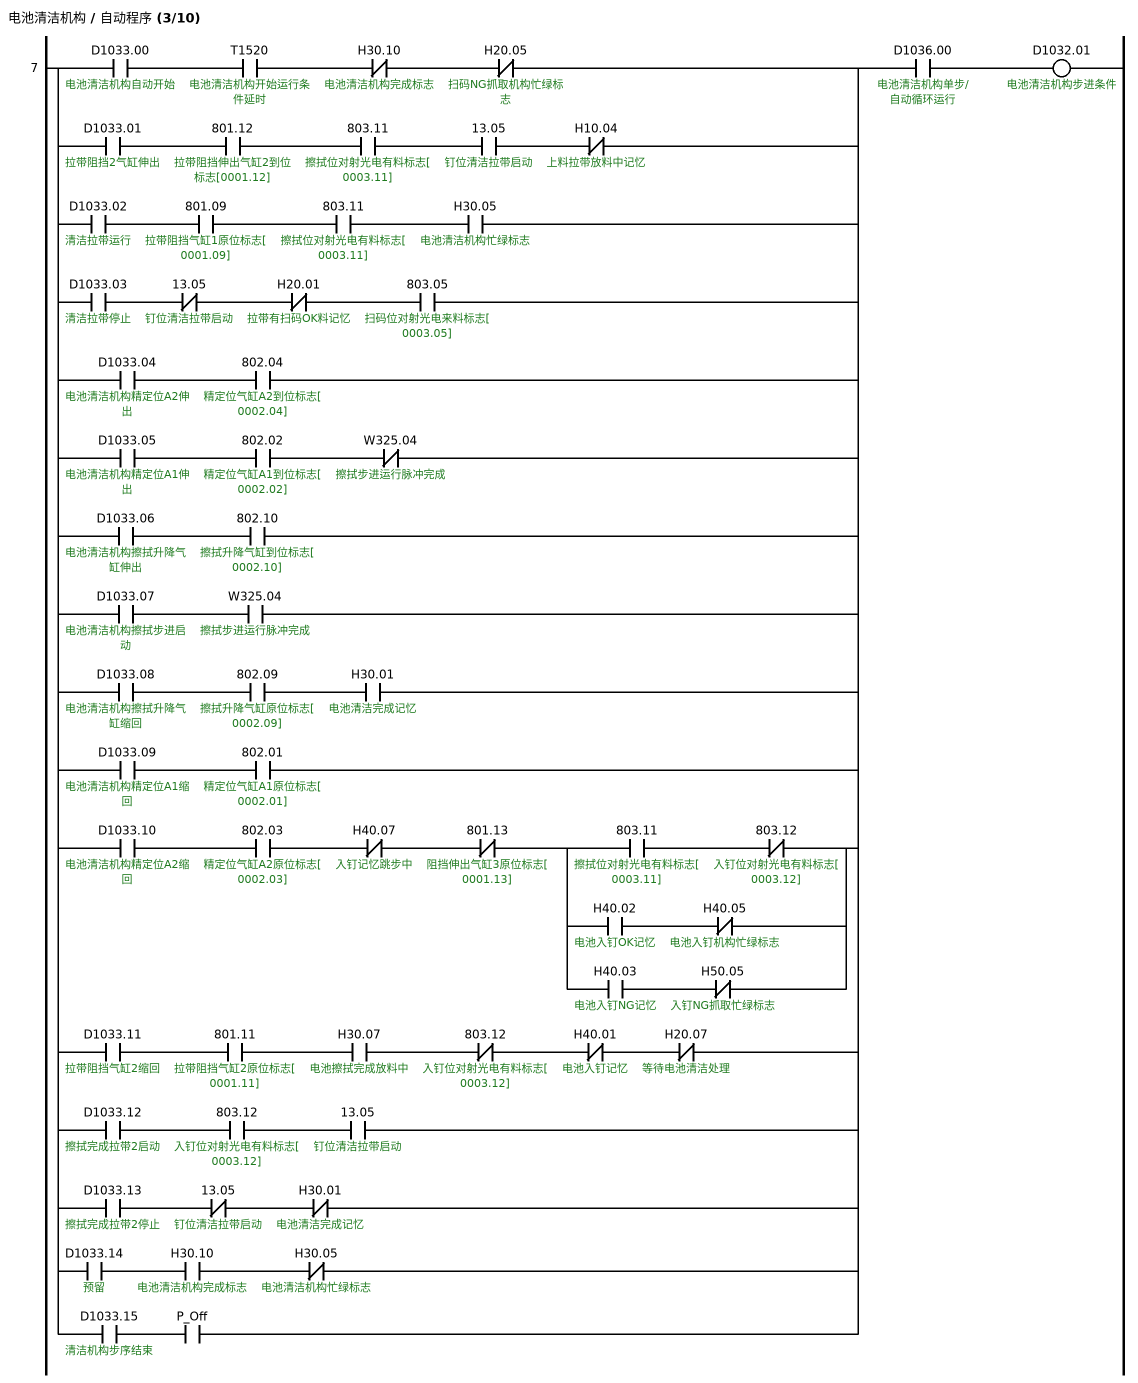
; rung 7
LD D1033.00  ; 电池清洁机构自动开始
AND T1520  ; 电池清洁机构开始运行条件延时
ANDNOT H30.10  ; 电池清洁机构完成标志
ANDNOT H20.05  ; 扫码NG抓取机构忙绿标志
LD D1033.01  ; 拉带阻挡2气缸伸出
AND 801.12  ; 拉带阻挡伸出气缸2到位标志[0001.12]
AND 803.11  ; 擦拭位对射光电有料标志[0003.11]
AND 13.05  ; 钉位清洁拉带启动
ANDNOT H10.04  ; 上料拉带放料中记忆
ORLD
LD D1033.02  ; 清洁拉带运行
AND 801.09  ; 拉带阻挡气缸1原位标志[0001.09]
AND 803.11  ; 擦拭位对射光电有料标志[0003.11]
AND H30.05  ; 电池清洁机构忙绿标志
ORLD
LD D1033.03  ; 清洁拉带停止
ANDNOT 13.05  ; 钉位清洁拉带启动
ANDNOT H20.01  ; 拉带有扫码OK料记忆
AND 803.05  ; 扫码位对射光电来料标志[0003.05]
ORLD
LD D1033.04  ; 电池清洁机构精定位A2伸出
AND 802.04  ; 精定位气缸A2到位标志[0002.04]
ORLD
LD D1033.05  ; 电池清洁机构精定位A1伸出
AND 802.02  ; 精定位气缸A1到位标志[0002.02]
ANDNOT W325.04  ; 擦拭步进运行脉冲完成
ORLD
LD D1033.06  ; 电池清洁机构擦拭升降气缸伸出
AND 802.10  ; 擦拭升降气缸到位标志[0002.10]
ORLD
LD D1033.07  ; 电池清洁机构擦拭步进启动
AND W325.04  ; 擦拭步进运行脉冲完成
ORLD
LD D1033.08  ; 电池清洁机构擦拭升降气缸缩回
AND 802.09  ; 擦拭升降气缸原位标志[0002.09]
AND H30.01  ; 电池清洁完成记忆
ORLD
LD D1033.09  ; 电池清洁机构精定位A1缩回
AND 802.01  ; 精定位气缸A1原位标志[0002.01]
ORLD
LD D1033.10  ; 电池清洁机构精定位A2缩回
AND 802.03  ; 精定位气缸A2原位标志[0002.03]
ANDNOT H40.07  ; 入钉记忆跳步中
ANDNOT 801.13  ; 阻挡伸出气缸3原位标志[0001.13]
LD 803.11  ; 擦拭位对射光电有料标志[0003.11]
ANDNOT 803.12  ; 入钉位对射光电有料标志[0003.12]
LD H40.02  ; 电池入钉OK记忆
ANDNOT H40.05  ; 电池入钉机构忙绿标志
ORLD
LD H40.03  ; 电池入钉NG记忆
ANDNOT H50.05  ; 入钉NG抓取忙绿标志
ORLD
ANDLD
ORLD
LD D1033.11  ; 拉带阻挡气缸2缩回
AND 801.11  ; 拉带阻挡气缸2原位标志[0001.11]
AND H30.07  ; 电池擦拭完成放料中
ANDNOT 803.12  ; 入钉位对射光电有料标志[0003.12]
ANDNOT H40.01  ; 电池入钉记忆
ANDNOT H20.07  ; 等待电池清洁处理
ORLD
LD D1033.12  ; 擦拭完成拉带2启动
AND 803.12  ; 入钉位对射光电有料标志[0003.12]
AND 13.05  ; 钉位清洁拉带启动
ORLD
LD D1033.13  ; 擦拭完成拉带2停止
ANDNOT 13.05  ; 钉位清洁拉带启动
ANDNOT H30.01  ; 电池清洁完成记忆
ORLD
LD D1033.14  ; 预留
AND H30.10  ; 电池清洁机构完成标志
ANDNOT H30.05  ; 电池清洁机构忙绿标志
ORLD
LD D1033.15  ; 清洁机构步序结束
AND P_Off
ORLD
AND D1036.00  ; 电池清洁机构单步/自动循环运行
OUT D1032.01  ; 电池清洁机构步进条件

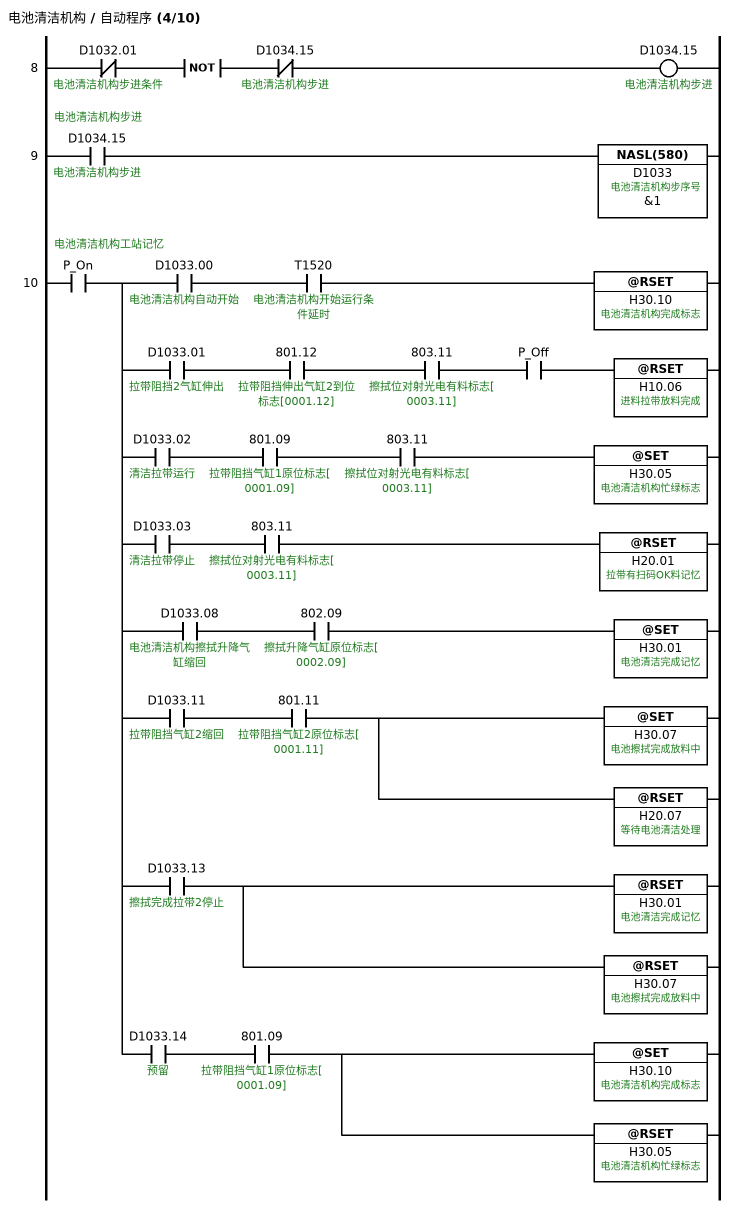
; rung 8
LDNOT D1032.01  ; 电池清洁机构步进条件
NOT(520)
ANDNOT D1034.15  ; 电池清洁机构步进
OUT D1034.15  ; 电池清洁机构步进
; rung 9: 电池清洁机构步进
LD D1034.15  ; 电池清洁机构步进
NASL(580) D1033 &1  ; 电池清洁机构步序号
; rung 10: 电池清洁机构工站记忆
LD P_On
OUT TR0
AND D1033.00  ; 电池清洁机构自动开始
AND T1520  ; 电池清洁机构开始运行条件延时
@RSET H30.10  ; 电池清洁机构完成标志
LD TR0
AND D1033.01  ; 拉带阻挡2气缸伸出
AND 801.12  ; 拉带阻挡伸出气缸2到位标志[0001.12]
AND 803.11  ; 擦拭位对射光电有料标志[0003.11]
AND P_Off
@RSET H10.06  ; 进料拉带放料完成
LD TR0
AND D1033.02  ; 清洁拉带运行
AND 801.09  ; 拉带阻挡气缸1原位标志[0001.09]
AND 803.11  ; 擦拭位对射光电有料标志[0003.11]
@SET H30.05  ; 电池清洁机构忙绿标志
LD TR0
AND D1033.03  ; 清洁拉带停止
AND 803.11  ; 擦拭位对射光电有料标志[0003.11]
@RSET H20.01  ; 拉带有扫码OK料记忆
LD TR0
AND D1033.08  ; 电池清洁机构擦拭升降气缸缩回
AND 802.09  ; 擦拭升降气缸原位标志[0002.09]
@SET H30.01  ; 电池清洁完成记忆
LD TR0
AND D1033.11  ; 拉带阻挡气缸2缩回
AND 801.11  ; 拉带阻挡气缸2原位标志[0001.11]
@SET H30.07  ; 电池擦拭完成放料中
@RSET H20.07  ; 等待电池清洁处理
LD TR0
AND D1033.13  ; 擦拭完成拉带2停止
@RSET H30.01  ; 电池清洁完成记忆
@RSET H30.07  ; 电池擦拭完成放料中
LD TR0
AND D1033.14  ; 预留
AND 801.09  ; 拉带阻挡气缸1原位标志[0001.09]
@SET H30.10  ; 电池清洁机构完成标志
@RSET H30.05  ; 电池清洁机构忙绿标志

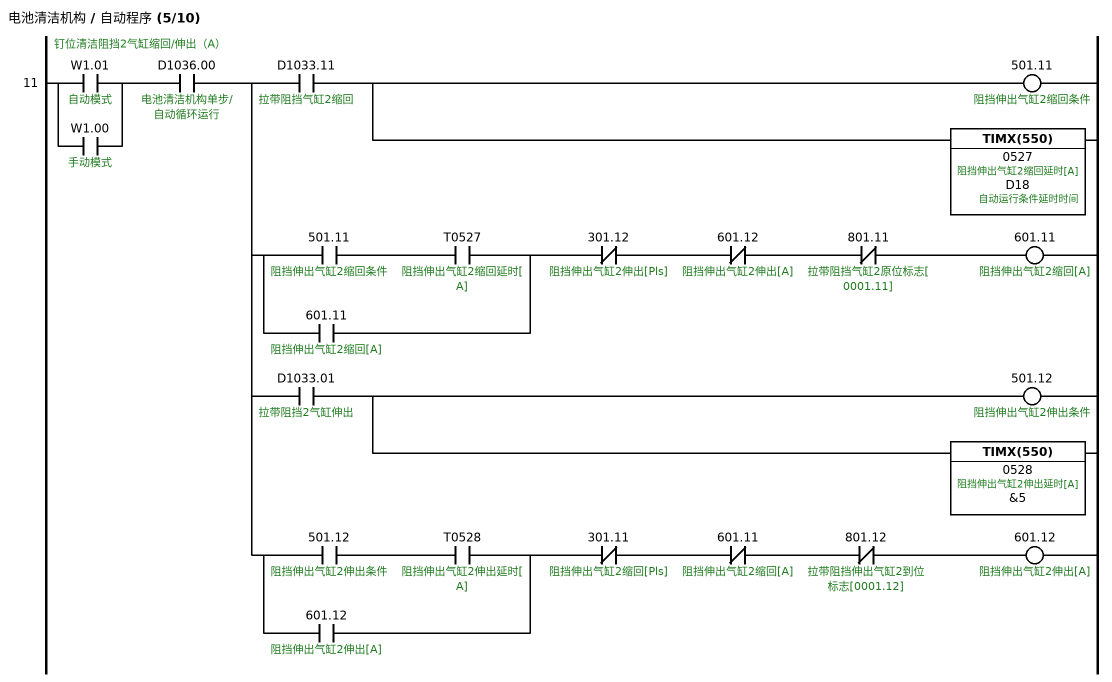
; rung 11: 钉位清洁阻挡2气缸缩回/伸出（A）
LD W1.01  ; 自动模式
OR W1.00  ; 手动模式
AND D1036.00  ; 电池清洁机构单步/自动循环运行
OUT TR0
AND D1033.11  ; 拉带阻挡气缸2缩回
OUT 501.11  ; 阻挡伸出气缸2缩回条件
TIMX(550) 0527 D18  ; 自动运行条件延时时间, 阻挡伸出气缸2缩回延时[A]
LD TR0
LD 501.11  ; 阻挡伸出气缸2缩回条件
AND T0527  ; 阻挡伸出气缸2缩回延时[A]
OR 601.11  ; 阻挡伸出气缸2缩回[A]
ANDLD
ANDNOT 301.12  ; 阻挡伸出气缸2伸出[Pls]
ANDNOT 601.12  ; 阻挡伸出气缸2伸出[A]
ANDNOT 801.11  ; 拉带阻挡气缸2原位标志[0001.11]
OUT 601.11  ; 阻挡伸出气缸2缩回[A]
LD TR0
AND D1033.01  ; 拉带阻挡2气缸伸出
OUT 501.12  ; 阻挡伸出气缸2伸出条件
TIMX(550) 0528 &5  ; 阻挡伸出气缸2伸出延时[A]
LD TR0
LD 501.12  ; 阻挡伸出气缸2伸出条件
AND T0528  ; 阻挡伸出气缸2伸出延时[A]
OR 601.12  ; 阻挡伸出气缸2伸出[A]
ANDLD
ANDNOT 301.11  ; 阻挡伸出气缸2缩回[Pls]
ANDNOT 601.11  ; 阻挡伸出气缸2缩回[A]
ANDNOT 801.12  ; 拉带阻挡伸出气缸2到位标志[0001.12]
OUT 601.12  ; 阻挡伸出气缸2伸出[A]

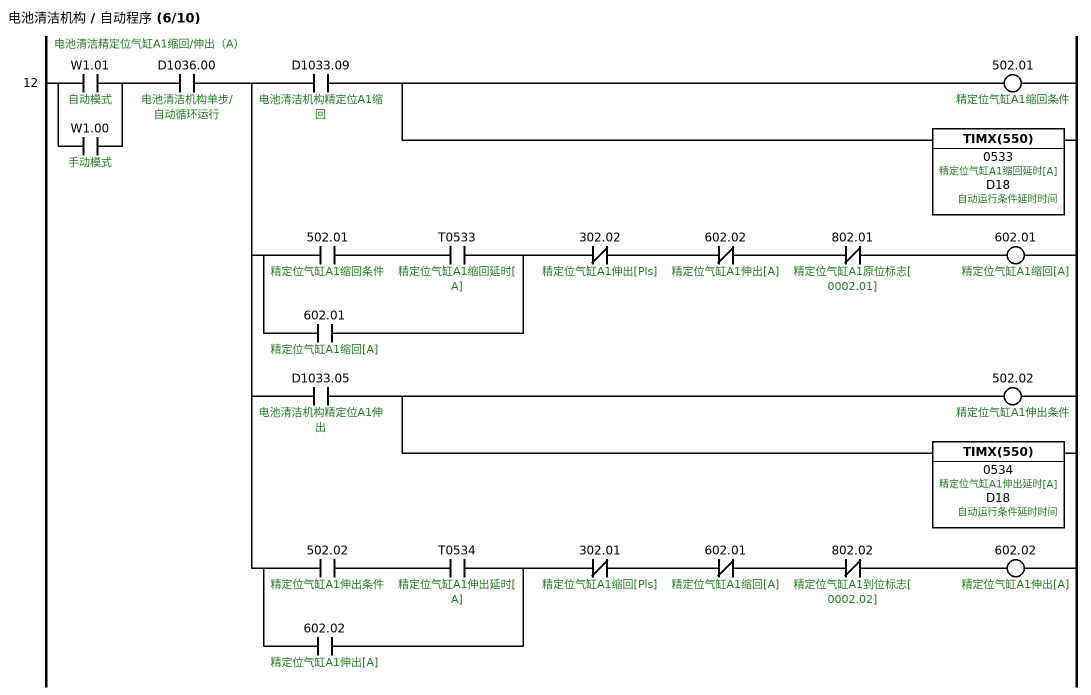
; rung 12: 电池清洁精定位气缸A1缩回/伸出（A）
LD W1.01  ; 自动模式
OR W1.00  ; 手动模式
AND D1036.00  ; 电池清洁机构单步/自动循环运行
OUT TR0
AND D1033.09  ; 电池清洁机构精定位A1缩回
OUT 502.01  ; 精定位气缸A1缩回条件
TIMX(550) 0533 D18  ; 自动运行条件延时时间, 精定位气缸A1缩回延时[A]
LD TR0
LD 502.01  ; 精定位气缸A1缩回条件
AND T0533  ; 精定位气缸A1缩回延时[A]
OR 602.01  ; 精定位气缸A1缩回[A]
ANDLD
ANDNOT 302.02  ; 精定位气缸A1伸出[Pls]
ANDNOT 602.02  ; 精定位气缸A1伸出[A]
ANDNOT 802.01  ; 精定位气缸A1原位标志[0002.01]
OUT 602.01  ; 精定位气缸A1缩回[A]
LD TR0
AND D1033.05  ; 电池清洁机构精定位A1伸出
OUT 502.02  ; 精定位气缸A1伸出条件
TIMX(550) 0534 D18  ; 自动运行条件延时时间, 精定位气缸A1伸出延时[A]
LD TR0
LD 502.02  ; 精定位气缸A1伸出条件
AND T0534  ; 精定位气缸A1伸出延时[A]
OR 602.02  ; 精定位气缸A1伸出[A]
ANDLD
ANDNOT 302.01  ; 精定位气缸A1缩回[Pls]
ANDNOT 602.01  ; 精定位气缸A1缩回[A]
ANDNOT 802.02  ; 精定位气缸A1到位标志[0002.02]
OUT 602.02  ; 精定位气缸A1伸出[A]

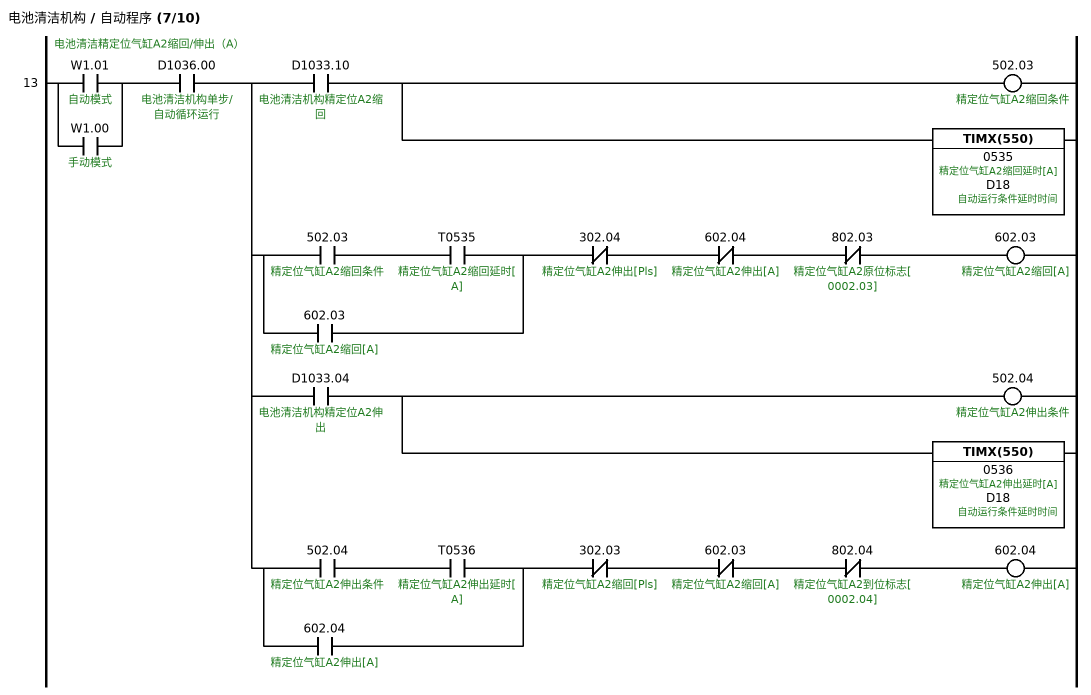
; rung 13: 电池清洁精定位气缸A2缩回/伸出（A）
LD W1.01  ; 自动模式
OR W1.00  ; 手动模式
AND D1036.00  ; 电池清洁机构单步/自动循环运行
OUT TR0
AND D1033.10  ; 电池清洁机构精定位A2缩回
OUT 502.03  ; 精定位气缸A2缩回条件
TIMX(550) 0535 D18  ; 自动运行条件延时时间, 精定位气缸A2缩回延时[A]
LD TR0
LD 502.03  ; 精定位气缸A2缩回条件
AND T0535  ; 精定位气缸A2缩回延时[A]
OR 602.03  ; 精定位气缸A2缩回[A]
ANDLD
ANDNOT 302.04  ; 精定位气缸A2伸出[Pls]
ANDNOT 602.04  ; 精定位气缸A2伸出[A]
ANDNOT 802.03  ; 精定位气缸A2原位标志[0002.03]
OUT 602.03  ; 精定位气缸A2缩回[A]
LD TR0
AND D1033.04  ; 电池清洁机构精定位A2伸出
OUT 502.04  ; 精定位气缸A2伸出条件
TIMX(550) 0536 D18  ; 自动运行条件延时时间, 精定位气缸A2伸出延时[A]
LD TR0
LD 502.04  ; 精定位气缸A2伸出条件
AND T0536  ; 精定位气缸A2伸出延时[A]
OR 602.04  ; 精定位气缸A2伸出[A]
ANDLD
ANDNOT 302.03  ; 精定位气缸A2缩回[Pls]
ANDNOT 602.03  ; 精定位气缸A2缩回[A]
ANDNOT 802.04  ; 精定位气缸A2到位标志[0002.04]
OUT 602.04  ; 精定位气缸A2伸出[A]

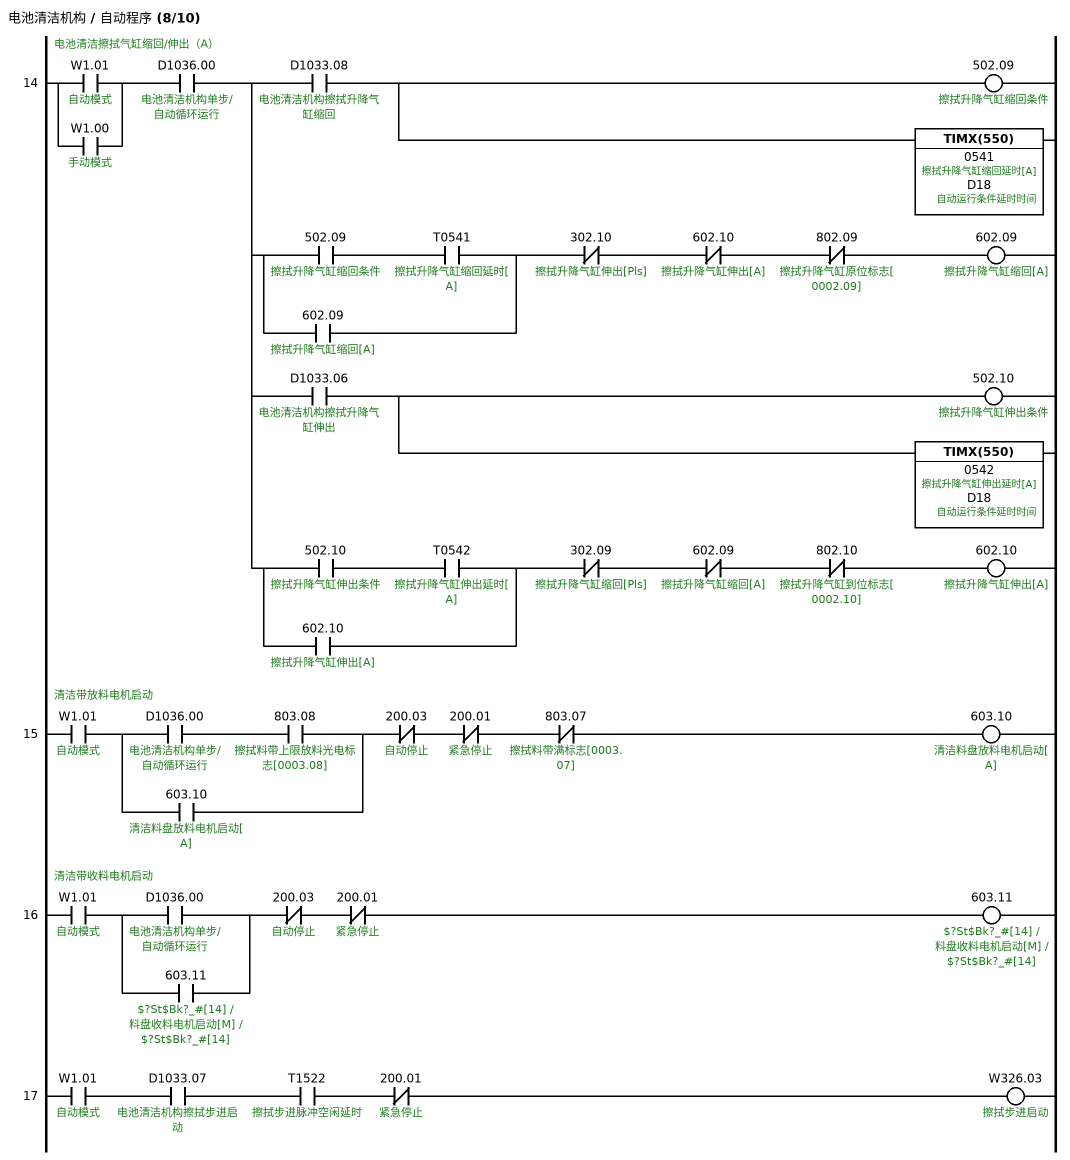
; rung 14: 电池清洁擦拭气缸缩回/伸出（A）
LD W1.01  ; 自动模式
OR W1.00  ; 手动模式
AND D1036.00  ; 电池清洁机构单步/自动循环运行
OUT TR0
AND D1033.08  ; 电池清洁机构擦拭升降气缸缩回
OUT 502.09  ; 擦拭升降气缸缩回条件
TIMX(550) 0541 D18  ; 自动运行条件延时时间, 擦拭升降气缸缩回延时[A]
LD TR0
LD 502.09  ; 擦拭升降气缸缩回条件
AND T0541  ; 擦拭升降气缸缩回延时[A]
OR 602.09  ; 擦拭升降气缸缩回[A]
ANDLD
ANDNOT 302.10  ; 擦拭升降气缸伸出[Pls]
ANDNOT 602.10  ; 擦拭升降气缸伸出[A]
ANDNOT 802.09  ; 擦拭升降气缸原位标志[0002.09]
OUT 602.09  ; 擦拭升降气缸缩回[A]
LD TR0
AND D1033.06  ; 电池清洁机构擦拭升降气缸伸出
OUT 502.10  ; 擦拭升降气缸伸出条件
TIMX(550) 0542 D18  ; 自动运行条件延时时间, 擦拭升降气缸伸出延时[A]
LD TR0
LD 502.10  ; 擦拭升降气缸伸出条件
AND T0542  ; 擦拭升降气缸伸出延时[A]
OR 602.10  ; 擦拭升降气缸伸出[A]
ANDLD
ANDNOT 302.09  ; 擦拭升降气缸缩回[Pls]
ANDNOT 602.09  ; 擦拭升降气缸缩回[A]
ANDNOT 802.10  ; 擦拭升降气缸到位标志[0002.10]
OUT 602.10  ; 擦拭升降气缸伸出[A]
; rung 15: 清洁带放料电机启动
LD W1.01  ; 自动模式
LD D1036.00  ; 电池清洁机构单步/自动循环运行
AND 803.08  ; 擦拭料带上限放料光电标志[0003.08]
OR 603.10  ; 清洁料盘放料电机启动[A]
ANDLD
ANDNOT 200.03  ; 自动停止
ANDNOT 200.01  ; 紧急停止
ANDNOT 803.07  ; 擦拭料带满标志[0003.07]
OUT 603.10  ; 清洁料盘放料电机启动[A]
; rung 16: 清洁带收料电机启动
LD W1.01  ; 自动模式
LD D1036.00  ; 电池清洁机构单步/自动循环运行
OR 603.11  ; $?St$Bk?_#[14] / 料盘收料电机启动[M] / $?St$Bk?_#[14]
ANDLD
ANDNOT 200.03  ; 自动停止
ANDNOT 200.01  ; 紧急停止
OUT 603.11  ; $?St$Bk?_#[14] / 料盘收料电机启动[M] / $?St$Bk?_#[14]
; rung 17
LD W1.01  ; 自动模式
AND D1033.07  ; 电池清洁机构擦拭步进启动
AND T1522  ; 擦拭步进脉冲空闲延时
ANDNOT 200.01  ; 紧急停止
OUT W326.03  ; 擦拭步进启动

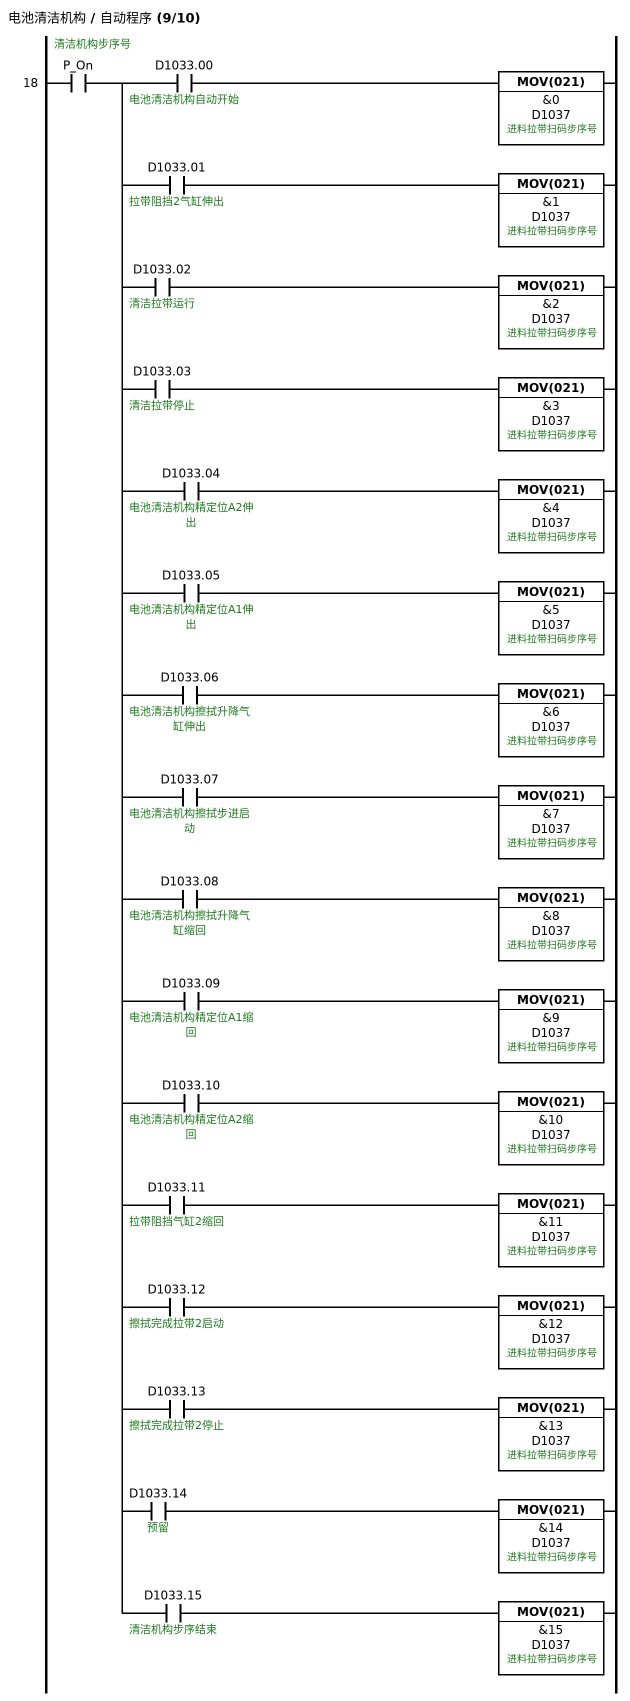
; rung 18: 清洁机构步序号
LD P_On
OUT TR0
AND D1033.00  ; 电池清洁机构自动开始
MOV(021) &0 D1037  ; 进料拉带扫码步序号
LD TR0
AND D1033.01  ; 拉带阻挡2气缸伸出
MOV(021) &1 D1037  ; 进料拉带扫码步序号
LD TR0
AND D1033.02  ; 清洁拉带运行
MOV(021) &2 D1037  ; 进料拉带扫码步序号
LD TR0
AND D1033.03  ; 清洁拉带停止
MOV(021) &3 D1037  ; 进料拉带扫码步序号
LD TR0
AND D1033.04  ; 电池清洁机构精定位A2伸出
MOV(021) &4 D1037  ; 进料拉带扫码步序号
LD TR0
AND D1033.05  ; 电池清洁机构精定位A1伸出
MOV(021) &5 D1037  ; 进料拉带扫码步序号
LD TR0
AND D1033.06  ; 电池清洁机构擦拭升降气缸伸出
MOV(021) &6 D1037  ; 进料拉带扫码步序号
LD TR0
AND D1033.07  ; 电池清洁机构擦拭步进启动
MOV(021) &7 D1037  ; 进料拉带扫码步序号
LD TR0
AND D1033.08  ; 电池清洁机构擦拭升降气缸缩回
MOV(021) &8 D1037  ; 进料拉带扫码步序号
LD TR0
AND D1033.09  ; 电池清洁机构精定位A1缩回
MOV(021) &9 D1037  ; 进料拉带扫码步序号
LD TR0
AND D1033.10  ; 电池清洁机构精定位A2缩回
MOV(021) &10 D1037  ; 进料拉带扫码步序号
LD TR0
AND D1033.11  ; 拉带阻挡气缸2缩回
MOV(021) &11 D1037  ; 进料拉带扫码步序号
LD TR0
AND D1033.12  ; 擦拭完成拉带2启动
MOV(021) &12 D1037  ; 进料拉带扫码步序号
LD TR0
AND D1033.13  ; 擦拭完成拉带2停止
MOV(021) &13 D1037  ; 进料拉带扫码步序号
LD TR0
AND D1033.14  ; 预留
MOV(021) &14 D1037  ; 进料拉带扫码步序号
LD TR0
AND D1033.15  ; 清洁机构步序结束
MOV(021) &15 D1037  ; 进料拉带扫码步序号

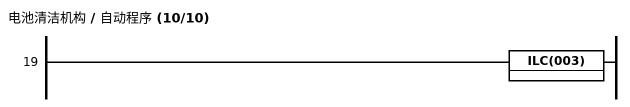
; rung 19
ILC(003)

### Section 状态指示灯

